(* Logix 5000 project; controller RSL5k_18_Template_noLib Emulate 5570 rev 32.11; software revision 32.02 *)
// Template Application with only task layout pre-installed

TASK _Controller_Status (periodic, rate 250 ms, priority 15, watchdog 2000 ms) : Diagnostics   // L_CPU, etc., and checks for Process Tasks that are Inhibited -- DO NOT INHIBIT THIS TASK
TASK Task_A_50ms (periodic, rate 50 ms, priority 5, watchdog 150 ms) : Task_A_MainProgram   // 50ms period Task
TASK Task_B_100ms (periodic, rate 100 ms, priority 6, watchdog 300 ms) : Task_B_MainProgram   // 100ms period Task
TASK Task_C_250ms (periodic, rate 250 ms, priority 7, watchdog 750 ms) : Task_C_MainProgram   // 250ms period Task
TASK Task_D_500ms (periodic, rate 500 ms, priority 8, watchdog 1500 ms) : Tank1   // 500ms period Task
TASK Task_E_1s (periodic, rate 1000 ms, priority 9, watchdog 3000 ms) : Task_E_MainProgram   // 1000ms (1s) period Task
TASK Task_F_2s (periodic, rate 2000 ms, priority 10, watchdog 6000 ms) : Task_F_MainProgram   // 2000ms (2s) period Task
TASK Task_G_5s (periodic, rate 5000 ms, priority 11, watchdog 15000 ms) : Task_G_MainProgram   // 5000ms (5s) period Task
TASK Task_H_10s (periodic, rate 10000 ms, priority 12, watchdog 30000 ms) : Task_H_MainProgram   // 10000ms (10s) period Task

MODULES
   Local : Emulate 5570 (ICP 2, rev 32.11)
END_MODULES

TYPE P_DescList :   // Code / Description List Entry
STRUCT
   Code : DINT;   // Code for which to look up Description
   Desc : STRING_40;   // Description for given Code
END_STRUCT
END_TYPE

TYPE STRING_12 :
STRUCT
   LEN : DINT;
   DATA : SINT[12];
END_STRUCT
END_TYPE

TYPE STRING_16 :
STRUCT
   LEN : DINT;
   DATA : SINT[16];
END_STRUCT
END_TYPE

TYPE STRING_20 :
STRUCT
   LEN : DINT;
   DATA : SINT[20];
END_STRUCT
END_TYPE

TYPE STRING_40 :
STRUCT
   LEN : DINT;
   DATA : SINT[40];
END_STRUCT
END_TYPE

TYPE STRING_8 :
STRUCT
   LEN : DINT;
   DATA : SINT[8];
END_STRUCT
END_TYPE

TYPE STRING_Area :
STRUCT
   LEN : DINT;
   DATA : SINT[8];
END_STRUCT
END_TYPE

TYPE STRING_Cond :
STRUCT
   LEN : DINT;
   DATA : SINT[20];
END_STRUCT
END_TYPE

TYPE STRING_NavTag :   // Navigation Tag
STRUCT
   LEN : DINT;
   DATA : SINT[20];
END_STRUCT
END_TYPE

ADD_ON_INSTRUCTION JLB_FopdtSim   (* revision 1.0 *)
VAR_INPUT
   cv : REAL; {visible}
   gain : REAL := 1.0; {visible}
   deadTime : REAL := 2.0; {visible}
   timeConst : REAL := 10.0; {visible}
END_VAR
VAR_OUTPUT
   pv : REAL; {access Read Only, visible}
END_VAR
VAR_INPUT
   pvss : REAL; {visible}
   cvss : REAL; {visible}
   pvLimitLow : REAL; {visible}
   pvLimitHigh : REAL := 100.0; {visible}
END_VAR
VAR
   DEDT1 : DEADTIME := (Gain := 1.0, RTSTime := 1);
   LDLG_01 : LEAD_LAG := (Gain := 1.0, RTSTime := 1);
   DEDT1_Array : REAL[500]; {access None}
   SUB_01 : FBD_MATH; {access None}
   HLL_01 : HL_LIMIT; {access None}
   pvUnlimited : REAL; {access None}
   initHigh : REAL; {access None}
   initLow : REAL; {access None}
   LDLG_Limiter_01 : JLB_LdlgLimiter; {access None}
   __l8BF204123A1F2166 : REAL; {access None}
   __l48C57120F21BA85D : REAL; {access None}
   __l0C3A629CB0B0CE2E : REAL; {access None}
   __l3C5358207E677F0D : REAL; {access None}
   __lCAFA7742E4AD4225 : REAL; {access None}
   __lA52B1C482AF3A637 : REAL; {access None}
   __l3430A9F65FF7AABD : REAL; {access None}
   __l4977D2FAECBF782C : REAL; {access None}
   __lBE5B6059D0DA292D : REAL; {access None}
END_VAR

ROUTINE Logic   (* function block diagram *)
   SHEET 1
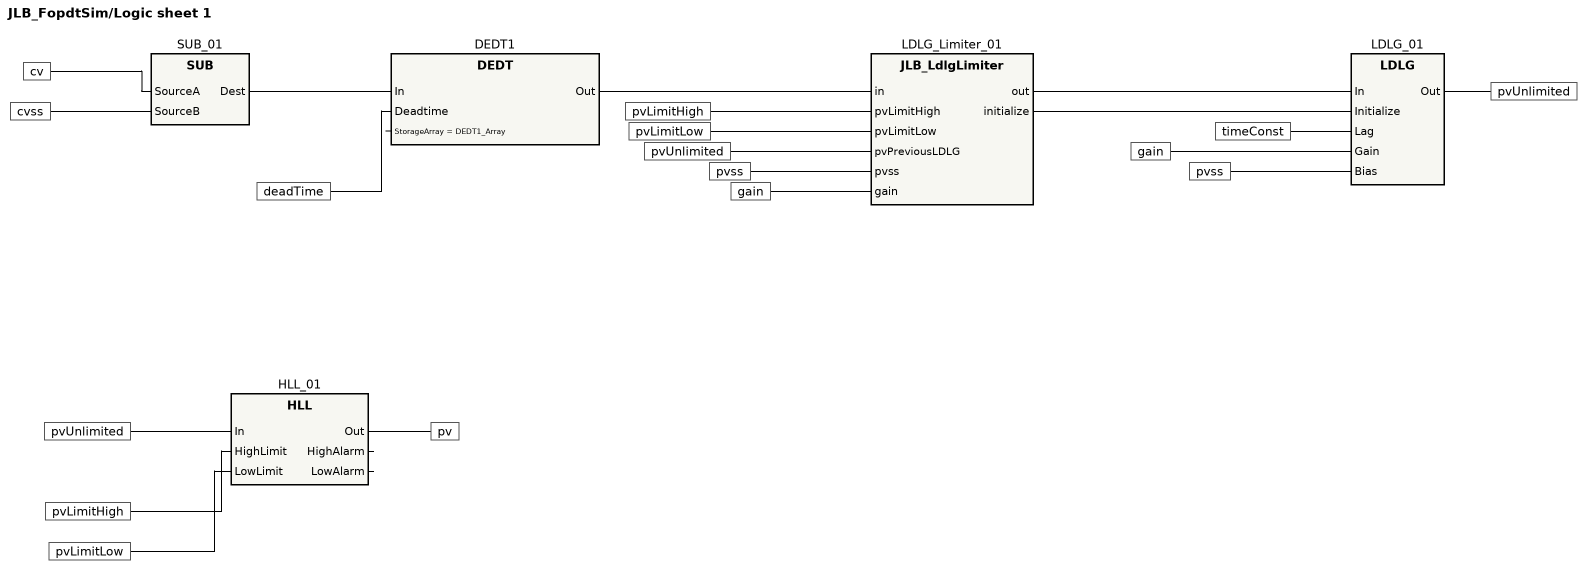
   SUB_01 : SUB(SourceA := cv, SourceB := cvss);
   HLL_01 : HLL(In := pvUnlimited, HighLimit := pvLimitHigh, LowLimit := pvLimitLow);   // unwired pins: HighAlarm LowAlarm
   DEDT1 : DEDT(In := SUB_01.Dest, Deadtime := deadTime, StorageArray := DEDT1_Array);
   pv := HLL_01.Out;
   LDLG_Limiter_01 : JLB_LdlgLimiter(in := DEDT1.Out, pvLimitHigh := pvLimitHigh, pvLimitLow := pvLimitLow, pvPreviousLDLG := pvUnlimited, pvss := pvss, gain := gain);
   LDLG_01 : LDLG(In := LDLG_Limiter_01.out, Initialize := LDLG_Limiter_01.initialize, Lag := timeConst, Gain := gain, Bias := pvss);
   pvUnlimited := LDLG_01.Out;
END_ROUTINE
END_ADD_ON_INSTRUCTION

ADD_ON_INSTRUCTION JLB_IpdtSim   (* revision 1.0 *)
VAR_INPUT
   cv : REAL; {required}
   gain : REAL; {visible}
   deadTime : REAL; {visible}
END_VAR
VAR_OUTPUT
   pv : REAL; {access Read Only, visible}
END_VAR
VAR_INPUT
   cvss : REAL;
   pvLimitHigh : REAL; {visible}
   pvLimitLow : REAL; {visible}
END_VAR
VAR
   DEDT1 : DEADTIME := (Gain := 1.0, RTSTime := 1);
   DEDT1_Array : REAL[500]; {access None}
   SUB_01 : FBD_MATH; {access None}
   INTG_01 : INTEGRATOR := (RTSTime := 1); {access None}
   __lDA04D48D4FBD5F02 : REAL; {access None}
   __lEF2A4DA27C9E24B0 : REAL; {access None}
   __l6744ED6412311BD7 : REAL; {access None}
   __lC3B18D60DF270F58 : REAL; {access None}
   __lFBECCCE1573B33CA : REAL; {access None}
   __lD020E224334B7143 : REAL; {access None}
END_VAR

ROUTINE Logic   (* function block diagram *)
   SHEET 1
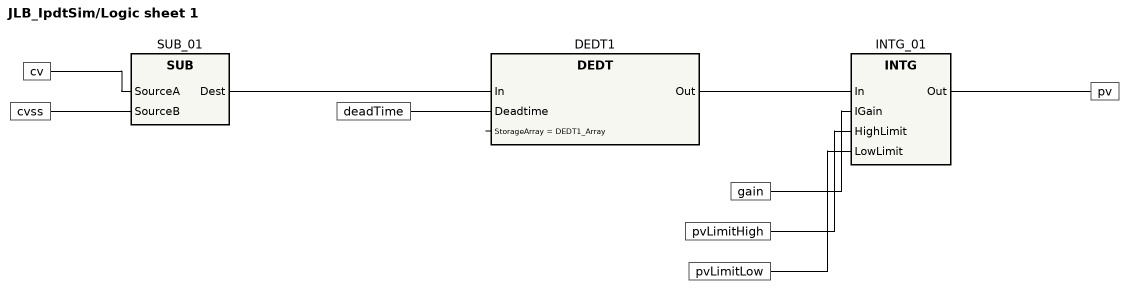
   SUB_01 : SUB(SourceA := cv, SourceB := cvss);
   DEDT1 : DEDT(In := SUB_01.Dest, Deadtime := deadTime, StorageArray := DEDT1_Array);
   INTG_01 : INTG(In := DEDT1.Out, IGain := gain, HighLimit := pvLimitHigh, LowLimit := pvLimitLow);
   pv := INTG_01.Out;
END_ROUTINE
END_ADD_ON_INSTRUCTION

ADD_ON_INSTRUCTION JLB_LdlgLimiter   (* revision 1.0 *)
// Reinitializes a LDLG.Out value to a limit value when limits are exceeded
VAR_INPUT
   in : REAL; {required}   // Normal Process Input
   pvLimitHigh : REAL; {visible}
   pvLimitLow : REAL; {visible}
   pvPreviousLDLG : REAL; {required}   // previous LDLG.Out
   pvss : REAL; {visible}
   gain : REAL; {visible}
END_VAR
VAR_OUTPUT
   out : REAL; {access Read Only, required}   // to LDLG.In
   initialize : BOOL; {access Read Only, visible}   // to LDLG.Initialize
END_VAR
VAR
   initHigh : REAL; {access Read Only}
   initLow : REAL; {access Read Only}
END_VAR

ROUTINE Logic   (* ladder *)
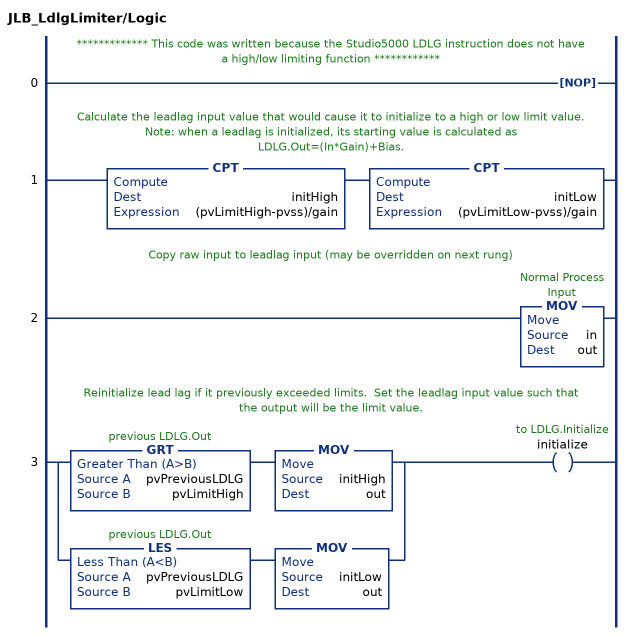
   // ************* This code was written because the Studio5000 LDLG instruction does not have a high/low limiting function ************
   0: NOP();
   // Calculate the leadlag input value that would cause it to initialize to a high or low limit value.
   // Note: when a leadlag is initialized, its starting value is calculated as LDLG.Out=(In*Gain)+Bias.
   1: CPT(initHigh,(pvLimitHigh-pvss)/gain)CPT(initLow,(pvLimitLow-pvss)/gain);
   // Copy raw input to leadlag input (may be overridden on next rung)
   2: MOV(in,out);
   // Reinitialize lead lag if it previously exceeded limits.  Set the leadlag input value such that the output will be the limit value.
   3: [GRT(pvPreviousLDLG,pvLimitHigh) MOV(initHigh,out) ,LES(pvPreviousLDLG,pvLimitLow) MOV(initLow,out) ]OTE(initialize);
END_ROUTINE
END_ADD_ON_INSTRUCTION

ADD_ON_INSTRUCTION L_TaskMon   (* revision 4.10 .00 Release, vendor Rockwell Automation *)
// Logix Task Monitor
// Revision note:
// See Instruction Help for a summary of changes, and see 4.10 Release Notes for details.
// Help:
// Copyright © Rockwell Automation, Inc.  All Rights Reserved.
// This Instruction monitors the controller Task in which it is contained and provides:
// *  Display Values for Task configuration: Task Name, Priority, Rate, Watchdog settings
// *  Display Values for Task statistics: Last and Max Execution time, Overlap Count
// *  Display of the Task Inhibit / Active Status
// *  Configuration of a "Plan" Execution Time, the time in which the Task is expected
//      to always complete (including interrupts by higher priority Tasks)
// *  An optional Alarm when Last (actual) Execution Time exceeds Plan
// *  A Reset command, which clears and acknowledges the Over Plan Alarm.
// *  Maintenance Commands to clear the Max Execution Time and Overlap Count.
// *  A configurable single-letter Task Identifier (for HMI)
// SUMMARY OF CHANGES FROM PREVIOUS VERSION (4.00.00)
// See 4.10 Release Notes for details.
// * Unmodified, up-rev only for Library 4.10.00
// SUMMARY OF CHANGES FROM PREVIOUS VERSION (3.5-01)
// See 4.00 Release Notes for details.
// * Changed Inf_ items to HMI_, and added Cfg_Area for security.
// * Deleted Cfg_PCmdClear; all Program Commands are now self-clearing.
// * Aligned ready bit naming with command bit names.
// * Removed unused STRING Local Tags.
// * All OCmds/MCmds and ORdys/MRdys are now Local Tags.
// * Added Sts_RdyAck and Sts_RdyReset for use by external objects.
VAR_INPUT
   Inp_Reset : BOOL; {visible}   // 1=Reset Max Task Time and any Alarm requiring reset
   Cfg_HasOverPlanAlm : ALIAS FOR OverPlan.Cfg_Exists;   // 1=Task Plan Exceeded Alarm exists and will be checked
   Cfg_OverPlanResetReqd : ALIAS FOR OverPlan.Cfg_ResetReqd;   // 1=Task Plan Exceeded Alarm is latched in, requires Reset Command to clear
   Cfg_OverPlanAckReqd : ALIAS FOR OverPlan.Cfg_AckReqd;   // 1=Task Plan Exceeded Alarm must be acknowledged
   Cfg_OverPlanSeverity : ALIAS FOR OverPlan.Cfg_Severity;   // Task Plan Exceeded Alarm Severity: 1=low, 2=medium, 3=high, 4=highest
   Cfg_PlanExecT : REAL := 3000.0;   // Expected Execution Time of Task (including interrupts) (ms)
   PCmd_Reset : BOOL;   // Program Command to Reset latched Alarm and Max Task Time
   PCmd_OverPlanAck : ALIAS FOR OverPlan.PCmd_Reset;   // Program Command to Acknowledge the Task Plan Exceeded Alarm
   PCmd_OverPlanSuppress : ALIAS FOR OverPlan.PCmd_Suppress;   // Program Command to Inhibit the Task Plan Exceeded Alarm
   PCmd_OverPlanUnsuppress : ALIAS FOR OverPlan.PCmd_Unsuppress;   // Program Command to Uninhibit the Task Plan Exceeded Alarm
   PCmd_OverPlanUnshelve : ALIAS FOR OverPlan.PCmd_Unshelve;   // Program Command to Unshelve the Task Plan Exceeded Alarm
END_VAR
VAR_OUTPUT
   Val_Rate : REAL; {access Read Only, visible}   // Configured Task Period (ms)
   Val_Priority : DINT; {access Read Only, visible}   // Configured Task Priority (1..15, lower number is higher priority)
   Val_LastExecT : REAL; {access Read Only, visible}   // Actual Last Execution Time of Task (ms)
   Val_MaxExecT : REAL; {access Read Only, visible}   // Highest Execution Time of Task (ms)
   Val_OverlapC : DINT; {access Read Only, visible}   // Task Overlap Count
   Val_WatchdogT : REAL; {access Read Only, visible}   // Configured Task Watchdog Timer Value (ms)
   Val_NotifyAll : DINT; {access Read Only}   // Highest Alarm prio and ack status this object + channel (enum)
   Val_UnackAlmC : DINT; {access Read Only}   // Count of Unacknowledged Alarms
   Sts_TaskInhibited : BOOL; {access Read Only, visible}   // 1=Task is Inhibited, 0 = Task is Active
   Sts_AlmInh : BOOL; {access Read Only}   // 1=An Alarm is Shelved, Disabled or Suppressed: display icon
   Sts_Err : BOOL; {access Read Only, visible}   // 1=Error in Config: see detail bits for reason
   Err_Plan : BOOL; {access Read Only}   // 1=Error in Config: Task Planned Exec Time (use 0.1 to 20,000.0 ms)
   Err_Alarm : BOOL; {access Read Only}   // 1=Error in Config: Alarm Min On Time or Severity
   Sts_RdyReset : ALIAS FOR ORdy_Reset; {access Read Only}   // 1=A latched alarm or shed condition is ready to be reset
   Sts_RdyAck : BOOL; {access Read Only}   // 1=An alarm is ready to be acknowledged
   Sts_OverPlan : ALIAS FOR OverPlan.Inp; {visible}   // 1=Task Actual Time exceeds Plan Time
   Alm_OverPlan : ALIAS FOR OverPlan.Alm;   // 1=Alarm: Planned Task Time Exceeded
   Ack_OverPlan : ALIAS FOR OverPlan.Ack;   // 1=Task Plan Exceeded Alarm has been acknowledged
   Sts_OverPlanDisabled : ALIAS FOR OverPlan.Disabled;   // 1=Task Plan Exceeded Alarm has been Disabled by Maintenance
   Sts_OverPlanSuppressed : ALIAS FOR OverPlan.Suppressed;   // 1=Task Plan Exceeded Alarm has been Suppressed by Program
   Sts_OverPlanShelved : ALIAS FOR OverPlan.Shelved;   // 1=Task Plan Exceeded Alarm has been Shelved by Operator
   L_TaskMon : BOOL;   // Unique Parameter Name for auto - discovery
END_VAR
VAR
   OverPlan : P_Alarm := (Inp := 1, Cfg_Exists := 1, Cfg_AckReqd := 1, Cfg_AllowShelve := 1, Cfg_AllowDisable := 1, Cfg_Severity := 750, Cfg_AlmMinOnT := 5, PCfg_AllowExist := 1, Ack := 1);   // Alarm if Actual Task Execution Time exceeds Planned
   Wrk_Inhibited : DINT; {access None}   // Task Inhibited if nonzero, Active if zero
   Val_Name : STRING_40; {access Read Only}   // Task Name as configured in Controller
   Wrk_Rate : DINT; {access None}   // Task Configured Rate (Period) from GSV (us)
   Wrk_LastExecT : DINT; {access None}   // Task Last Execution Time from GSV (us)
   Wrk_MaxExecT : DINT; {access None}   // Task Maximum Execution Time from GSV (us)
   Wrk_WatchdogT : DINT; {access None}   // Task Configured Watchdog Time from GSV (us)
   HMI_Tab : SINT;   // Tab to display (FTView ME)
   Wrk_Notify : DINT; {access None}   // Buffer for building Val_Notify
   Val_Notify : DINT; {access Read Only}   // Current Alarm Level and Acknowledgement (enumeration)
   HMI_Type : STRING_16 := 'L_TaskMon'; {access Read Only}   // Must contain AOI name, used for HMI and Information S/W
   Cfg_Area : STRING_Area := 'area01';   // Process Area for security
   HMI_Lib : STRING_12 := 'RA-BAS'; {access Read Only}   // Display Library for Faceplate call-up
   Wrk_UnackAlmC : DINT; {access None}   // Buffer for building Val_UnackAlmC
   ORdy_ResetAckAll : BOOL; {access Read Only}   // 1=At least one Alarm requires Reset or Acknowledgement
   ORdy_Reset : BOOL; {access Read Only}   // 1=Ready for OCmd_Reset (enables button)
   OCmd_ResetAckAll : BOOL;   // Operator Command to Reset and Acknowledge all Alarms
   OCmd_Reset : BOOL;   // Operator Command to Reset latched Alarm and Max Task Time
   MCmd_ClearOverlapC : BOOL;   // Maintenance Command to Clear Task Overlap Count
   MCmd_ClearMaxExecT : BOOL;   // Maintenance Command to Clear Maximum Execution Time
END_VAR

ROUTINE Logic   (* ladder *)
// Monitor the Task containing this AOI and alarm if over planned scan time.
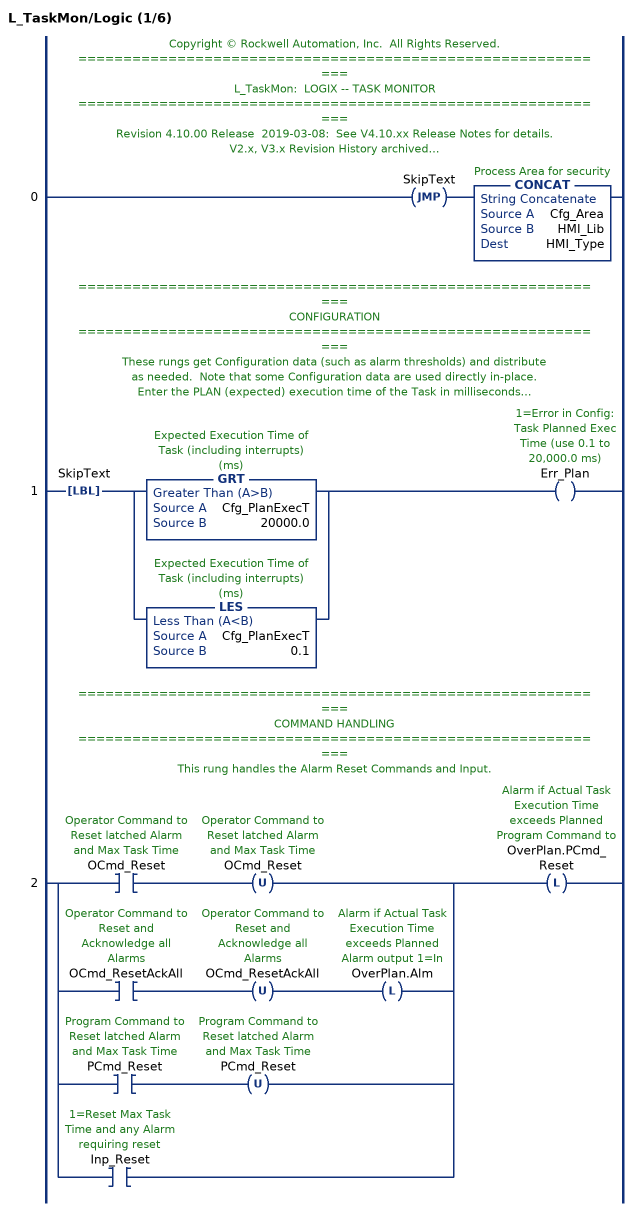
   // Copyright © Rockwell Automation, Inc.  All Rights Reserved.
   // ============================================================
   // L_TaskMon:  LOGIX -- TASK MONITOR
   // ============================================================
   // Revision 4.10.00 Release  2019-03-08:  See V4.10.xx Release Notes for details.
   // V2.x, V3.x Revision History archived.
   // V4.00.00  2018-06-19:  Changed Inf_ items to HMI_ and added Cfg_Area for security.
   // Added unacked alarm count. Deleted Cfg_PCmdClear; all Program
   // Commands are now self-clearing. Aligned ready bit naming with
   // command bit names. Removed unused STRING Local Tags.
   // All OCmds/MCmds and ORdys/MRdys are now Local Tags.
   // Added Sts_RdyAck and Sts_ResetReqd for use by external objects.
   // V4.10.00  2019-03-08:  Unmodified, up-rev only for Library 4.10.00
   // ============================================================
   // This Instruction monitors the controller Task in which it is contained
   // and provides:
   // *  Display Values for Task configuration: Task Name, Priority, Rate, Watchdog settings
   // *  Display Values for Task statistics: Last and Max Execution time, Overlap Count
   // *  Display of the Task Inhibit / Active Status
   // *  Configuration of a "Plan" Execution Time, the time in which the Task is expected
   //  to always complete (including interrupts by higher priority Tasks)
   // *  An optional Alarm when Last (actual) Execution Time exceeds Plan
   // *  A Reset command, which clears and acknowledges the Over Plan Alarm.
   // *  Maintenance Commands to clear the Max Execution Time and Overlap Count.
   // *  A configurable single-letter Task Identifier (for HMI)
   // ============================================================
   // SHOW LOCAL STRINGS
   // ============================================================
   // The STRINGs containing the text associated with each instance of this
   // instruction cannot be Input or Output Parameters, because STRINGs are not
   //  'atomic' types. (Inputs and Outputs must be SINT, INT, DINT, REAL, or BOOL.)
   // In order to make it easier to find and configure these STRINGs, this rung
   // was added.  THE JMP (and the LBL on the following rung)
   // MUST NOT BE REMOVED!!!
   // To view the STRINGs, go to the instruction instance (in LD or FBD), RIGHT-click
   // to bring up the context menu and select "Open Instruction Logic".
   // This rung will appear with the STRING values for the selected instance.
   // You may double-click the STRING values here to modify them as well.
   // #####  V4.00.00  2018-06-19:  Added string for Cfg_Area, renamed Inf_* to HMI_*,  #####
   // #####  removed unused STRING Local Tags.  #####
   0: JMP(SkipText)CONCAT(Cfg_Area,HMI_Lib,HMI_Type);
   // ============================================================
   // CONFIGURATION
   // ============================================================
   // These rungs get Configuration data (such as alarm thresholds) and distribute
   // as needed.  Note that some Configuration data are used directly in-place.
   // Enter the PLAN (expected) execution time of the Task in milliseconds.
   // If the actual execution time of the Task (which includes interrupts by higher priority
   // Tasks) exceeds this threshold, the OverPlan Status is raised
   // (and the OverPlan Alarm is raised if so configured).
   1: LBL(SkipText)[GRT(Cfg_PlanExecT,20000.0) ,LES(Cfg_PlanExecT,0.1) ]OTE(Err_Plan);
   // ============================================================
   // COMMAND HANDLING
   // ============================================================
   // This rung handles the Alarm Reset Commands and Input.
   2: [XIC(OCmd_Reset) OTU(OCmd_Reset) ,XIC(OCmd_ResetAckAll) OTU(OCmd_ResetAckAll) OTL(OverPlan.Alm) ,XIC(PCmd_Reset) OTU(PCmd_Reset) ,XIC(Inp_Reset) ]OTL(OverPlan.PCmd_Reset);
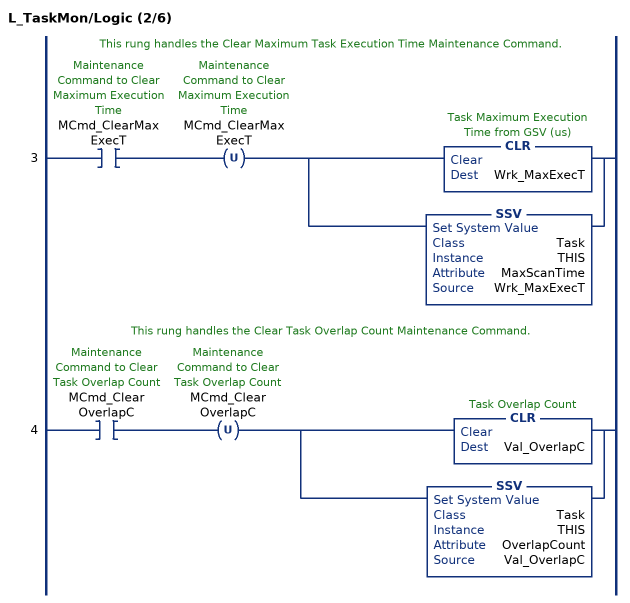
   // This rung handles the Clear Maximum Task Execution Time Maintenance Command.
   3: XIC(MCmd_ClearMaxExecT)OTU(MCmd_ClearMaxExecT)[CLR(Wrk_MaxExecT) ,SSV(Task,THIS,MaxScanTime,Wrk_MaxExecT) ];
   // This rung handles the Clear Task Overlap Count Maintenance Command.
   4: XIC(MCmd_ClearOverlapC)OTU(MCmd_ClearOverlapC)[CLR(Val_OverlapC) ,SSV(Task,THIS,OverlapCount,Val_OverlapC) ];
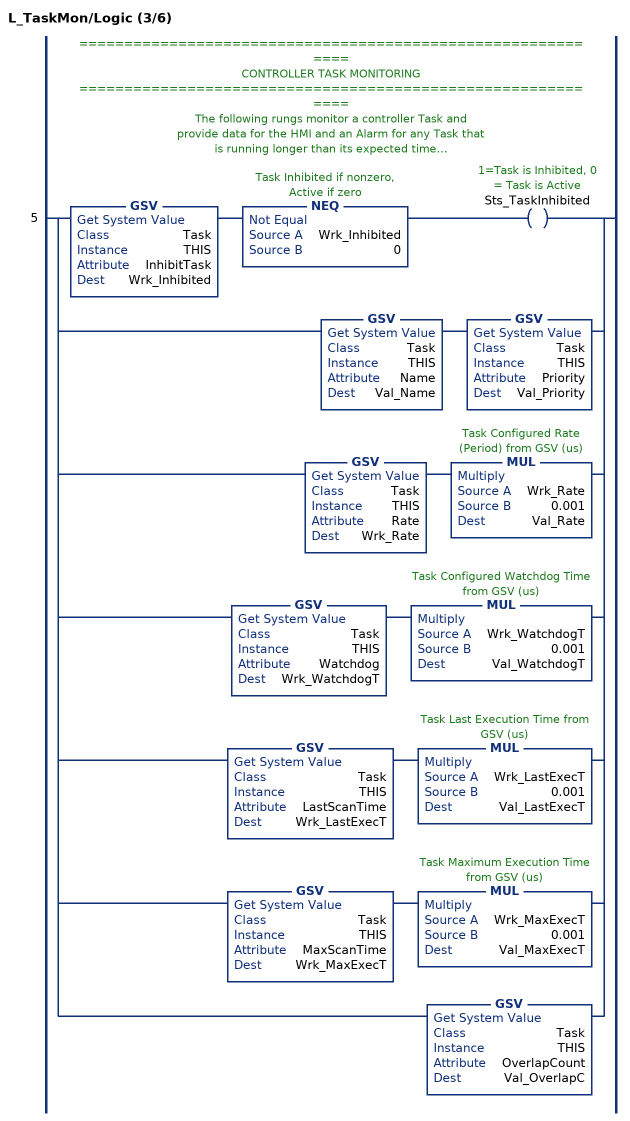
   // ============================================================
   // CONTROLLER TASK MONITORING
   // ============================================================
   // The following rungs monitor a controller Task and
   // provide data for the HMI and an Alarm for any Task that
   // is running longer than its expected time.
   // This rung provides the following Task configuration data:
   // * Task Inhibited status
   // * Task Name
   // * Task Priority
   // * Task Period (Rate) (ms)
   // * Task Watchdog Timeout setting (ms)
   // ... and provides the following Task statistics:
   // * Task Last Execution Time (ms)
   // * Task Maximum Execution Time (ms)
   // * Task Overlap Count
   5: [GSV(Task,THIS,InhibitTask,Wrk_Inhibited) NEQ(Wrk_Inhibited,0) OTE(Sts_TaskInhibited) ,GSV(Task,THIS,Name,Val_Name) GSV(Task,THIS,Priority,Val_Priority) ,GSV(Task,THIS,Rate,Wrk_Rate) MUL(Wrk_Rate,0.001,Val_Rate) ,GSV(Task,THIS,Watchdog,Wrk_WatchdogT) MUL(Wrk_WatchdogT,0.001,Val_WatchdogT) ,GSV(Task,THIS,LastScanTime,Wrk_LastExecT) MUL(Wrk_LastExecT,0.001,Val_LastExecT) ,GSV(Task,THIS,MaxScanTime,Wrk_MaxExecT) MUL(Wrk_MaxExecT,0.001,Val_MaxExecT) ,GSV(Task,THIS,OverlapCount,Val_OverlapC) ];
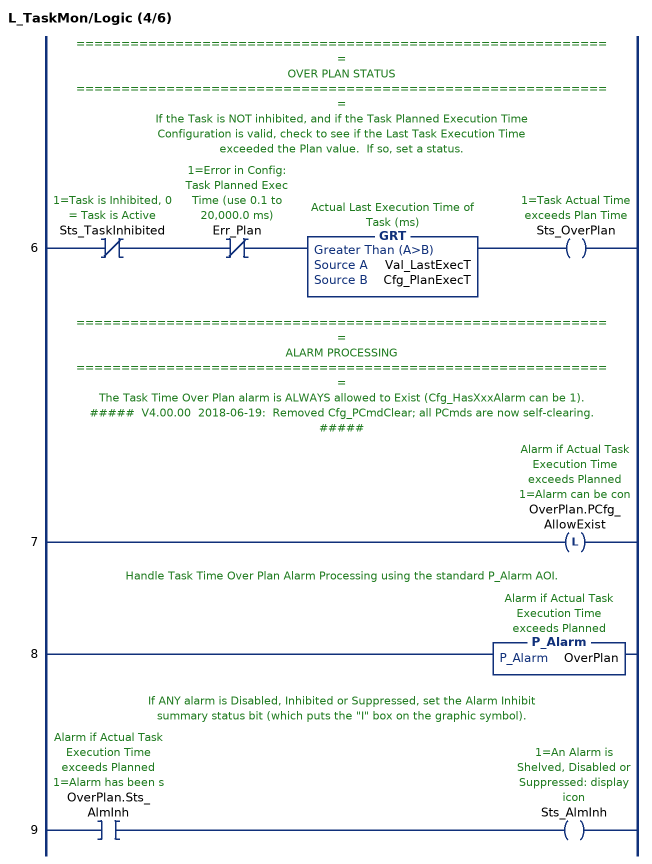
   // ============================================================
   // OVER PLAN STATUS
   // ============================================================
   // If the Task is NOT inhibited, and if the Task Planned Execution Time
   // Configuration is valid, check to see if the Last Task Execution Time
   // exceeded the Plan value.  If so, set a status.
   6: XIO(Sts_TaskInhibited)XIO(Err_Plan)GRT(Val_LastExecT,Cfg_PlanExecT)OTE(Sts_OverPlan);
   // ============================================================
   // ALARM PROCESSING
   // ============================================================
   // The Task Time Over Plan alarm is ALWAYS allowed to Exist (Cfg_HasXxxAlarm can be 1).
   // #####  V4.00.00  2018-06-19:  Removed Cfg_PCmdClear; all PCmds are now self-clearing.  #####
   7: OTL(OverPlan.PCfg_AllowExist);
   // Handle Task Time Over Plan Alarm Processing using the standard P_Alarm AOI.
   8: P_Alarm(OverPlan);
   // If ANY alarm is Disabled, Inhibited or Suppressed, set the Alarm Inhibit
   // summary status bit (which puts the "I" box on the graphic symbol).
   9: XIC(OverPlan.Sts_AlmInh)OTE(Sts_AlmInh);
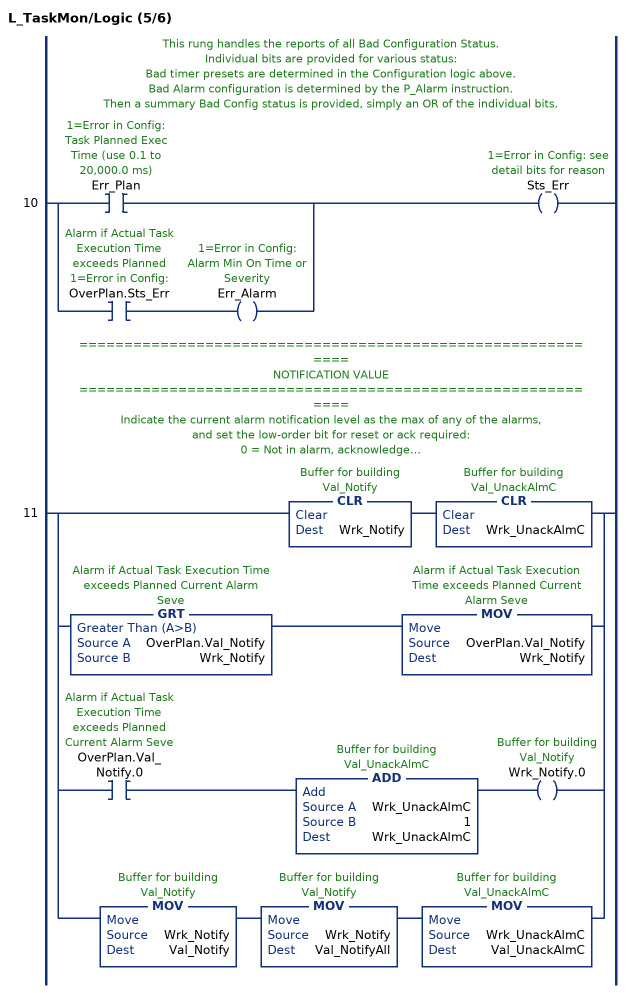
   // This rung handles the reports of all Bad Configuration Status.
   // Individual bits are provided for various status:
   // Bad timer presets are determined in the Configuration logic above.
   // Bad Alarm configuration is determined by the P_Alarm instruction.
   // Then a summary Bad Config status is provided, simply an OR of the individual bits.
   10: [XIC(Err_Plan) ,XIC(OverPlan.Sts_Err) OTE(Err_Alarm) ]OTE(Sts_Err);
   // ============================================================
   // NOTIFICATION VALUE
   // ============================================================
   // Indicate the current alarm notification level as the max of any of the alarms,
   // and set the low-order bit for reset or ack required:
   // 0 = Not in alarm, acknowledged
   // 1 = Not in alarm, unacknowledged or reset required
   // 2 = Low severity alarm, acknowledged
   // 3 = Low severity alarm, unacknowledged
   // 4 = Medium severity alarm, acknowledged
   // 5 = Medium severity alarm, unacknowledged
   // 6 = High severity alarm, acknowledged
   // 7 = High severity alarm, unacknowledged
   // 8 = Urgent severity alarm, acknowledged
   // 9 = Urgent severity alarm, unacknowledged
   // #####  V4.00.00  2018-06-19:  Added Val_NotifyAll and unacked alarm count.  #####
   11: [CLR(Wrk_Notify) CLR(Wrk_UnackAlmC) ,GRT(OverPlan.Val_Notify,Wrk_Notify) MOV(OverPlan.Val_Notify,Wrk_Notify) ,XIC(OverPlan.Val_Notify.0) ADD(Wrk_UnackAlmC,1,Wrk_UnackAlmC) OTE(Wrk_Notify.0) ,MOV(Wrk_Notify,Val_Notify) MOV(Wrk_Notify,Val_NotifyAll) MOV(Wrk_UnackAlmC,Val_UnackAlmC) ];
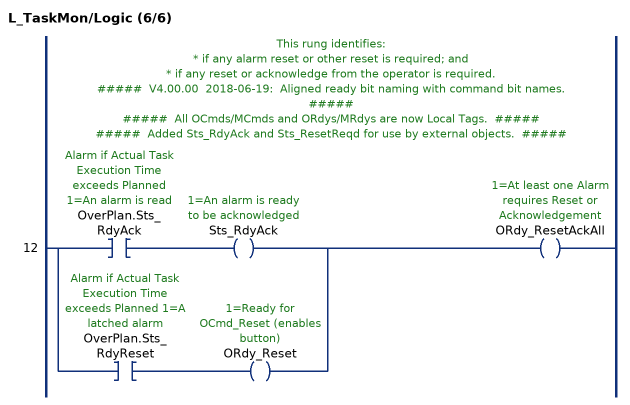
   // This rung identifies:
   // * if any alarm reset or other reset is required; and
   // * if any reset or acknowledge from the operator is required.
   // #####  V4.00.00  2018-06-19:  Aligned ready bit naming with command bit names.  #####
   // #####  All OCmds/MCmds and ORdys/MRdys are now Local Tags.  #####
   // #####  Added Sts_RdyAck and Sts_ResetReqd for use by external objects.  #####
   12: [XIC(OverPlan.Sts_RdyAck) OTE(Sts_RdyAck) ,XIC(OverPlan.Sts_RdyReset) OTE(ORdy_Reset) ]OTE(ORdy_ResetAckAll);
END_ROUTINE
END_ADD_ON_INSTRUCTION

ADD_ON_INSTRUCTION P_AIn   (* revision 4.10 .00 Release, vendor Rockwell Automation, ExecutePrescan, ExecuteEnableInFalse *)
// Analog Input
// Revision note:
// See Instruction Help for a summary of changes, and see 4.10 Release Notes for details.
// Help:
// Copyright © Rockwell Automation, Inc.  All Rights Reserved.
// This Instruction monitors an Analog Input from a flow, level, pressure,
// temperature, or any other analog sensor, and provides:
// *  Scaling, from Input (Raw) to PV (Engineering) Units
// *  High-High, High, Low and Low-Low Status and Alarms, with Gate
// inputs and configurable on-delay, off-delay and gate delay times
// *  Monitoring of bad/uncertain PV status, floating point exceptions
// and out-of-range conditions, with PV Fail alarm
// *  Setting of a simulated input signal for process simulation
// *  Capturing of the lowest and highest PV excursion values
// *  Configuration for status thresholds, deadbands and range limits
// *  Maintenance Commands to allow manual override of the input signal (Substitute PV)
// Alarms are provided by P_Alarm AOI instances.
// Status gating provided by P_Gate AOI instances.
// SUMMARY OF CHANGES FROM PREVIOUS VERSION (4.00.01)
// See 4.10 Release Notes for details.
// * Added Cfg_HasMoreObj.
// SUMMARY OF CHANGES FROM PREVIOUS VERSION (4.00.00)
// See 4.00 Release Notes for details.
// * Modified handling of SrcQ_IO and SrcQ.
// SUMMARY OF CHANGES FROM PREVIOUS VERSION (3.5-03)
// See 4.00 Release Notes for details.
// * Removed P_Mode, PSet/Val_Owner and related OSets,
//    PSets and Vals.  Thresholds are now Cfgs.
// * Changed Inf_ items to HMI_, and added Cfg_Area for security.
// * Added notify and unack count rollup for Channel object.
// * Changed Out-of-Range limit checks to use raw Input (Inp_PV)
//    instead of scaled PV (Val).  Changing EU scaling will not
//    necessitate changing fail thresholds and deadband.
// * Deleted Cfg_PCmdClear.  All Program Commands are now self-clearing.
// * Aligned ready bit naming with command bit names.
// * All OCmds/MCmds and ORdys/MRdys are now Local Tags.
// * Added Sts_RdyAck and Sts_RdyReset for use by external objects.
// * Removed Err_DB, code ensures Status Deadband configs are always valid.
// * Added configurable decimal places for display on HMI.
VAR_INPUT
   Inp_PV : REAL; {visible}   // Input Signal (process variable) from Sensor
   Inp_PVSrcQ : DINT;   // Input Source and Quality (from Channel object, if available) (enum)
   Inp_PVNotify : DINT;   // Related PV object alarm prio and ack status (enum)
   Inp_PVBad : BOOL;   // 1=PV or I/O Comms Status Bad, 0=OK
   Inp_PVUncertain : BOOL;   // 1=PV Value Not Reliable, 0=OK
   Inp_Sim : BOOL;   // 1=Use simulated PV (Set_SimPV); 0=Use Input (Inp_PV)
   Inp_HiHiGate : ALIAS FOR HiHiGate.Inp_Gate;   // High-High Status Gate, 1=enabled
   Inp_HiGate : ALIAS FOR HiGate.Inp_Gate;   // High Status Gate, 1=enabled
   Inp_LoGate : ALIAS FOR LoGate.Inp_Gate;   // Low Status Gate, 1=enabled
   Inp_LoLoGate : ALIAS FOR LoLoGate.Inp_Gate;   // Low-Low Status Gate, 1=enabled
   Inp_FailGate : ALIAS FOR FailGate.Inp_Gate;   // Fail Status Gate, 1=enabled
   Inp_Reset : BOOL;   // 1=Reset all Alarms requiring reset
   Cfg_NoSubstPV : BOOL;   // 1=Disallow selection of Substitute PV
   Cfg_HasChanObj : BOOL;   // 1=Tells HMI a Channel object (AIChan, etc.) is used for Inp_PV
   Cfg_HasMoreObj : BOOL;   // 1=Tells HMI an object with more info is available
   Cfg_UseChanSrcQ : BOOL;   // 1=Pass thru connected Channel's SrcQ value, 0=generate SrcQ
   Cfg_PVDecPlcs : DINT := 2;   // Number of decimal places for PV display (0..6)
   Cfg_HasHiHiAlm : ALIAS FOR HiHi.Cfg_Exists;   // 1=High-High Alarm exists and will be checked
   Cfg_HasHiAlm : ALIAS FOR Hi.Cfg_Exists;   // 1=High Alarm exists and will be checked
   Cfg_HasLoAlm : ALIAS FOR Lo.Cfg_Exists;   // 1=Low Alarm exists and will be checked
   Cfg_HasLoLoAlm : ALIAS FOR LoLo.Cfg_Exists;   // 1=Low-Low Alarm exists and will be checked
   Cfg_HasFailAlm : ALIAS FOR Fail.Cfg_Exists;   // 1=Analog Input Failure Alarm exists and will be checked
   Cfg_HiHiResetReqd : ALIAS FOR HiHi.Cfg_ResetReqd;   // 1=Reset required to clear High-High Alarm
   Cfg_HiResetReqd : ALIAS FOR Hi.Cfg_ResetReqd;   // 1=Reset required to clear High Alarm
   Cfg_LoResetReqd : ALIAS FOR Lo.Cfg_ResetReqd;   // 1=Reset required to clear Low Alarm
   Cfg_LoLoResetReqd : ALIAS FOR LoLo.Cfg_ResetReqd;   // 1=Reset required to clear Low-Low Alarm
   Cfg_FailResetReqd : ALIAS FOR Fail.Cfg_ResetReqd;   // 1=Reset required to clear Analog InputFailure Alarm
   Cfg_HiHiAckReqd : ALIAS FOR HiHi.Cfg_AckReqd;   // 1=Acknowledge required for High-High Alarm
   Cfg_HiAckReqd : ALIAS FOR Hi.Cfg_AckReqd;   // 1=Acknowledge required for High Alarm
   Cfg_LoAckReqd : ALIAS FOR Lo.Cfg_AckReqd;   // 1=Acknlowledge required for Low Alarm
   Cfg_LoLoAckReqd : ALIAS FOR LoLo.Cfg_AckReqd;   // 1=Acknowledge required for Low-Low Alarm
   Cfg_FailAckReqd : ALIAS FOR Fail.Cfg_AckReqd;   // 1=Acknowledge required for Analog Input Failure Alarm
   Cfg_HiHiSeverity : ALIAS FOR HiHi.Cfg_Severity;   // High-High Alarm Severity: 1..250=Low, 251..500=Medium, 501..750=High, 751..1000=Urgent
   Cfg_HiSeverity : ALIAS FOR Hi.Cfg_Severity;   // High Alarm Severity: 1..250=Low, 251..500=Medium, 501..750=High, 751..1000=Urgent
   Cfg_LoSeverity : ALIAS FOR Lo.Cfg_Severity;   // Low Alarm Severity: 1..250=Low, 251..500=Medium, 501..750=High, 751..1000=Urgent
   Cfg_LoLoSeverity : ALIAS FOR LoLo.Cfg_Severity;   // Low-Low Alarm Severity: 1..250=Low, 251..500=Medium, 501..750=High, 751..1000=Urgent
   Cfg_FailSeverity : ALIAS FOR Fail.Cfg_Severity;   // Failure Alarm Severity: 1..250=Low, 251..500=Medium, 501..750=High, 751..1000=Urgent
   Cfg_InpRawMin : REAL;   // Input (unscaled) Minimum for Scaling
   Cfg_InpRawMax : REAL := 100.0;   // Input (unscaled) Maximum for Scaling
   Cfg_PVEUMin : REAL;   // PV (Output) Minimum for Scaling to EU
   Cfg_PVEUMax : REAL := 100.0;   // PV (Output) Maximum for Scaling to EU
   Cfg_FiltTC : REAL;   // PV Filter Time Constant (s), 0.0 = unfiltered
   Cfg_HiHiLim : REAL := 1.5e+38; {visible}   // High-High Status Threshold (EU)
   Cfg_HiHiDB : REAL := 1.0;   // High-High Status Deadband (EU)
   Cfg_HiHiOnDly : ALIAS FOR HiHiGate.Cfg_OnDly;   // Minimum time above High-High Limit to raise Status (s)
   Cfg_HiHiOffDly : ALIAS FOR HiHiGate.Cfg_OffDly;   // Minimum time below High-High Limit (minus deadband) to clear Status (s)
   Cfg_HiHiGateDly : ALIAS FOR HiHiGate.Cfg_GateDly;   // High-High Status Gate Delay (s)
   Cfg_HiLim : REAL := 1.5e+38; {visible}   // High Status Threshold (EU)
   Cfg_HiDB : REAL := 1.0;   // High Status Deadband (EU)
   Cfg_HiOnDly : ALIAS FOR HiGate.Cfg_OnDly;   // Minimum time above High Limit to raise Status (s)
   Cfg_HiOffDly : ALIAS FOR HiGate.Cfg_OffDly;   // Minimum time below High Limit (minus deadband) to clear Status (s)
   Cfg_HiGateDly : ALIAS FOR HiGate.Cfg_GateDly;   // High Status Gate Delay (s)
   Cfg_LoLim : REAL := -1.5e+38; {visible}   // Low Status Threshold (EU)
   Cfg_LoDB : REAL := 1.0;   // Low Status Deadband (EU)
   Cfg_LoOnDly : ALIAS FOR LoGate.Cfg_OnDly;   // Minimum time below Low Limit to raise Status (s)
   Cfg_LoOffDly : ALIAS FOR LoGate.Cfg_OffDly;   // Minimum time above Low Limit (plus deadband) to clear Status (s)
   Cfg_LoGateDly : ALIAS FOR LoGate.Cfg_GateDly;   // Low Status Gate Delay (s)
   Cfg_LoLoLim : REAL := -1.5e+38; {visible}   // Low-Low Status Threshold (EU)
   Cfg_LoLoDB : REAL := 1.0;   // Low-Low Status Deadband (EU)
   Cfg_LoLoOnDly : ALIAS FOR LoLoGate.Cfg_OnDly;   // Minimum time below Low-Low Limit to raise Status (s)
   Cfg_LoLoOffDly : ALIAS FOR LoLoGate.Cfg_OffDly;   // Minimum time above Low-Low Limit (plus deadband) to clear Status (s)
   Cfg_LoLoGateDly : ALIAS FOR LoLoGate.Cfg_GateDly;   // Low-Low Status Gate Delay (s)
   Cfg_FailHiLim : REAL := 103.958336;   // Out-of-Range (fail) High Limit (raw units)
   Cfg_FailLoLim : REAL := -2.0833333;   // Out-of-Range (fail) Low Limit (raw units)
   Cfg_FailDB : REAL := 0.41666666;   // Out-of-Range (fail) High/Low Deadband (raw units)
   Cfg_FailOnDly : ALIAS FOR FailGate.Cfg_OnDly;   // Minimum time Bad or Out of Range to raise Fail Status (s)
   Cfg_FailOffDly : ALIAS FOR FailGate.Cfg_OffDly;   // Minimum time OK or In Range to clear Fail Status (s)
   Cfg_FailGateDly : ALIAS FOR FailGate.Cfg_GateDly;   // Fail Status Gate Delay (s)
   Set_SimPV : REAL;   // PV used in Simulation (Inp_Sim=1) (EU)
   PCmd_ClearCapt : BOOL;   // Program Command to Clear the captured min / max PV excursion values
   PCmd_Reset : BOOL;   // Program Command to Reset all Alarms requiring Reset
   PCmd_HiHiAck : ALIAS FOR HiHi.PCmd_Ack;   // Program Command to Acknowledge High-High Alarm
   PCmd_HiHiSuppress : ALIAS FOR HiHi.PCmd_Suppress;   // Program Command to Suppress High-High Alarm
   PCmd_HiHiUnsuppress : ALIAS FOR HiHi.PCmd_Unsuppress;   // Program Command to Unsuppress High-High Alarm
   PCmd_HiHiUnshelve : ALIAS FOR HiHi.PCmd_Unshelve;   // Program Command to Unshelve High-High Alarm
   PCmd_HiAck : ALIAS FOR Hi.PCmd_Ack;   // Program Command to Acknowledge High Alarm
   PCmd_HiSuppress : ALIAS FOR Hi.PCmd_Suppress;   // Program Command to Suppress High Alarm
   PCmd_HiUnsuppress : ALIAS FOR Hi.PCmd_Unsuppress;   // Program Command to Unsuppress High Alarm
   PCmd_HiUnshelve : ALIAS FOR Hi.PCmd_Unshelve;   // Program Command to Unshelve High Alarm
   PCmd_LoAck : ALIAS FOR Lo.PCmd_Ack;   // Program Command to Acknowledge Low Alarm
   PCmd_LoSuppress : ALIAS FOR Lo.PCmd_Suppress;   // Program Command to Suppress Low Alarm
   PCmd_LoUnsuppress : ALIAS FOR Lo.PCmd_Unsuppress;   // Program Command to Unsuppress Low Alarm
   PCmd_LoUnshelve : ALIAS FOR Lo.PCmd_Unshelve;   // Program Command to Unshelve Low Alarm
   PCmd_LoLoAck : ALIAS FOR LoLo.PCmd_Ack;   // Program Command to Acknowledge Low-Low Alarm
   PCmd_LoLoSuppress : ALIAS FOR LoLo.PCmd_Suppress;   // Program Command to Suppress Low-Low Alarm
   PCmd_LoLoUnsuppress : ALIAS FOR LoLo.PCmd_Unsuppress;   // Program Command to Unsuppress Low-Low Alarm
   PCmd_LoLoUnshelve : ALIAS FOR LoLo.PCmd_Unshelve;   // Program Command to Unshelve Low-Low Alarm
   PCmd_FailAck : ALIAS FOR Fail.PCmd_Ack;   // Program Command to Acknowldege Analog Input Failure Alarm
   PCmd_FailSuppress : ALIAS FOR Fail.PCmd_Suppress;   // Program Command to Suppress Analog Input Failure Alarm
   PCmd_FailUnsuppress : ALIAS FOR Fail.PCmd_Unsuppress;   // Program Command to Unsuppress Analog Input Failure Alarm
   PCmd_FailUnshelve : ALIAS FOR Fail.PCmd_Unshelve;   // Program Command to Unshelve Analog Input Failure Alarm
END_VAR
VAR_OUTPUT
   Val : REAL; {access Read Only, visible}   // Analog Value (after Substitute PV, if used)
   Val_InpPV : REAL; {access Read Only, visible}   // Analog Input Value (actual, before Substitute PV selection)
   Val_PVMinCapt : REAL := 1.5e+38; {access Read Only}   // Captured PV Minimum (excursion) since last cleared
   Val_PVMaxCapt : REAL := -1.5e+38; {access Read Only}   // Captured PV Maximum (excursion) since last cleared
   Val_PVEUMin : REAL; {access Read Only}   // Minimum of scaled range = MIN (Cfg_PVEUMin, Cfg_PVEUMax)
   Val_PVEUMax : REAL := 100.0; {access Read Only}   // Maximum of scaled range = MAX (Cfg_PVEUMin, Cfg_PVEUMax)
   SrcQ_IO : DINT; {access Read Only}   // Source and Quality of primary I/O (enumeration)
   SrcQ : DINT; {access Read Only}   // Source and Quality of primary Val/Sts (enumeration)
   Val_Fault : DINT; {access Read Only}   // Device Fault Status 0=none, 20=Lo, 21=Hi, 24=LoLo, 25=HiHi, 32=Fail, 34=CfgErr
   Val_NotifyAll : DINT; {access Read Only}   // Highest Alarm prio and ack status this object + channel (enum)
   Val_UnackAlmC : DINT; {access Read Only}   // Count of Unacknowledged Alarms
   Sts_SubstPV : BOOL; {access Read Only}   // 1=Using Substitute PV (overrides input), 0=Using live Input PV from device
   Sts_PVBad : BOOL; {access Read Only}   // 1=PV Bad quality or Out of Range
   Sts_PVUncertain : BOOL; {access Read Only}   // 1=PV Value is Uncertain (quality)
   Sts_MaintByp : BOOL; {access Read Only}   // 1=A Maintenance Bypass is Active, display icon
   Sts_AlmInh : BOOL; {access Read Only}   // 1=An Alarm is Shelved, Disabled or Suppressed: display icon
   Sts_Err : BOOL; {access Read Only, visible}   // 1=Error in Config (see detail Err_ bits for reason), display icon
   Err_Raw : BOOL; {access Read Only}   // 1=Error in Config: Raw Input Scaling Min = Max
   Err_EU : BOOL; {access Read Only}   // 1=Error in Config: Scaled EU Min = Max
   Err_Timer : BOOL; {access Read Only}   // 1=Error in Config: On Delay, Off Delay, Gate Delay Time Invalid (use 0 to 2147483 s)
   Err_Filt : BOOL; {access Read Only}   // 1=Error in Config: PV filter params (RateTime, TC)
   Err_Alarm : BOOL; {access Read Only}   // 1=Error in Config: Alarm Min On Time, Shelf Time, Severity
   Sts_RdyReset : ALIAS FOR ORdy_Reset; {access Read Only}   // 1=A latched alarm or shed condition is ready to be reset
   Sts_RdyAck : BOOL; {access Read Only}   // 1=An alarm is ready to be acknowledged
   Sts_HiHiCmp : ALIAS FOR HiHiGate.Inp;   // PV High-High comparison result 1=High-High
   Sts_HiHiGate : ALIAS FOR HiHiGate.Sts_Gate; {access Read Only}   // PV High-High Gate Delay Status, 1=done
   Sts_HiHi : ALIAS FOR HiHi.Inp; {visible}   // 1=Analog Input is above High-High limit
   Alm_HiHi : ALIAS FOR HiHi.Alm;   // 1=Analog Input is in High-High Alarm
   Ack_HiHi : ALIAS FOR HiHi.Ack;   // 1=High-High Alarm has been acknowledged
   Sts_HiHiDisabled : ALIAS FOR HiHi.Disabled;   // 1=High-High Alarm has been Disabled by Maintenancy
   Sts_HiHiSuppressed : ALIAS FOR HiHi.Suppressed;   // 1=High-High Alarm has been Suppressed by Program
   Sts_HiHiShelved : ALIAS FOR HiHi.Shelved;   // 1=High-High Alarm has been Shelved by Operator
   Sts_HiCmp : ALIAS FOR HiGate.Inp;   // PV High comparison result 1=High
   Sts_HiGate : ALIAS FOR HiGate.Sts_Gate; {access Read Only}   // PV High Gate Delay Status, 1=done
   Sts_Hi : ALIAS FOR Hi.Inp; {visible}   // 1=Analog Input is above High limit
   Alm_Hi : ALIAS FOR Hi.Alm;   // 1=Analog Input is in High Alarm
   Ack_Hi : ALIAS FOR Hi.Ack;   // 1=High Alarm has been acknowledged
   Sts_HiDisabled : ALIAS FOR Hi.Disabled;   // 1=High Alarm has been Disabled by Maintenance
   Sts_HiSuppressed : ALIAS FOR Hi.Suppressed;   // 1=High Alarm has been Suppressed by Program
   Sts_HiShelved : ALIAS FOR Hi.Shelved;   // 1=High Alarm has been Shelved by Operator
   Sts_LoCmp : ALIAS FOR LoGate.Inp;   // PV Low comparison result 1=Low
   Sts_LoGate : ALIAS FOR LoGate.Sts_Gate; {access Read Only}   // PV Low Gate Delay Status, 1=done
   Sts_Lo : ALIAS FOR Lo.Inp; {visible}   // 1=Analog Input is below Low limit
   Alm_Lo : ALIAS FOR Lo.Alm;   // 1=Analog Input is in Low Alarm
   Ack_Lo : ALIAS FOR Lo.Ack;   // 1=Low Alarm has been acknowledged
   Sts_LoDisabled : ALIAS FOR Lo.Disabled;   // 1=Low Alarm has been Disabled by Maintenance
   Sts_LoSuppressed : ALIAS FOR Lo.Suppressed;   // 1=Low Alarm has been Suppressed by Program
   Sts_LoShelved : ALIAS FOR Lo.Shelved;   // 1=Low Alarm has been Shelved by Operator
   Sts_LoLoCmp : ALIAS FOR LoLoGate.Inp;   // PV Low-Low comparison result 1=Low-Low
   Sts_LoLoGate : ALIAS FOR LoLoGate.Sts_Gate; {access Read Only}   // PV Low-Low Gate Delay Status, 1=done
   Sts_LoLo : ALIAS FOR LoLo.Inp; {visible}   // 1=Analog Input is below Low-Low limit
   Alm_LoLo : ALIAS FOR LoLo.Alm;   // 1=Analog Input is in Low-Low Alarm
   Ack_LoLo : ALIAS FOR LoLo.Ack;   // 1=Low-Low Alarm has been acknowledged
   Sts_LoLoDisabled : ALIAS FOR LoLo.Disabled;   // 1=Low-Low Alarm has been Disabled by Maintenance
   Sts_LoLoSuppressed : ALIAS FOR LoLo.Suppressed;   // 1=Low-Low Alarm has been Suppressed by Program
   Sts_LoLoShelved : ALIAS FOR LoLo.Shelved;   // 1=Low-Low Alarm has been Shelved by Operator
   Sts_FailCmp : ALIAS FOR FailGate.Inp;   // PV Fail comparison result 1=Out of Range
   Sts_FailGate : ALIAS FOR FailGate.Sts_Gate; {access Read Only}   // PV Fail Gate Delay Status, 1=done
   Sts_Fail : ALIAS FOR Fail.Inp; {visible}   // 1=Analog Input is Out of Range or PV Bad
   Alm_Fail : ALIAS FOR Fail.Alm;   // 1=Analog Input Failure Alarm (PV Bad or Out of Range)
   Ack_Fail : ALIAS FOR Fail.Ack;   // 1=Analog Input Failure Alarm has been acknowledged
   Sts_FailDisabled : ALIAS FOR Fail.Disabled;   // 1=Analog input Failure Alarm has been Disabled by Maintenance
   Sts_FailSuppressed : ALIAS FOR Fail.Suppressed;   // 1=Analog Input Failure Alarm has been Suppressed by Program
   Sts_FailShelved : ALIAS FOR Fail.Shelved; {visible}   // 1=Analog Input Failure Alarm has been Shelved by Operator
   P_AIn : BOOL;   // Unique Parameter Name for auto - discovery
END_VAR
VAR
   LoLo : P_Alarm := (Cfg_AckReqd := 1, Cfg_AllowShelve := 1, Cfg_AllowDisable := 1, Cfg_Severity := 750, Cfg_AlmMinOnT := 5, PCfg_AllowExist := 1, Ack := 1);   // Low-Low Alarm
   Lo : P_Alarm := (Cfg_AckReqd := 1, Cfg_AllowShelve := 1, Cfg_AllowDisable := 1, Cfg_Severity := 500, Cfg_AlmMinOnT := 5, PCfg_AllowExist := 1, Ack := 1);   // Low Alarm
   Hi : P_Alarm := (Cfg_AckReqd := 1, Cfg_AllowShelve := 1, Cfg_AllowDisable := 1, Cfg_Severity := 500, Cfg_AlmMinOnT := 5, PCfg_AllowExist := 1, Ack := 1);   // High Alarm
   HiHi : P_Alarm := (Cfg_AckReqd := 1, Cfg_AllowShelve := 1, Cfg_AllowDisable := 1, Cfg_Severity := 750, Cfg_AlmMinOnT := 5, PCfg_AllowExist := 1, Ack := 1);   // High-High Alarm
   Cfg_EU : STRING_8 := '%';   // Engineering Units for display on HMI
   Cfg_Tag : STRING_20 := 'P_AIn';   // Tagname for display on HMI
   Cfg_Label : STRING_20 := 'Analog Input';   // Label for graphic symbol displayed on HMI
   Cfg_Desc : STRING_40 := 'Analog Input';   // Description for display on HMI
   Fail : P_Alarm := (Cfg_AckReqd := 1, Cfg_AllowShelve := 1, Cfg_AllowDisable := 1, Cfg_Severity := 1000, Cfg_AlmMinOnT := 5, PCfg_AllowExist := 1, Ack := 1);   // Analog Input Failure Alarm (bad quality or out of range)
   Wrk_Notify : DINT; {access None}   // Buffer for building Val_Notify
   HMI_Tab : SINT;   // Tab to display (FTView ME)
   Wrk_Fault : DINT; {access None}   // Buffer for building Val_Fault
   Wrk_SrcQ : DINT; {access None}   // Register for building Source / Quality enumeration
   Wrk_SubstPV : BOOL; {access None}   // Internal flag: Using Substitute PV
   Wrk_UnfiltPV : REAL; {access None}   // Unfiltered PV, input to 1st order filter
   Wrk_Alpha : REAL; {access None}   // Filter multiplier = (1 / (1+TC/dT) )
   Wrk_ScanT : TIMER := (PRE := 2147483647); {access None}   // Scan Timer (milliseconds, always runs)
   Wrk_ScanTime : REAL; {access None}   // Time since this instance was last scanned
   Wrk_FiltPV : REAL; {access None}   // Filtered PV
   Wrk_ValidONS : BOOL; {access None}   // Selected PV goes from Infinite or Not a Number to VALID
   Wrk_SelPVDINT : DINT; {access None}   // Selected PV check for Infinite or Non A Number
   Wrk_SelPVInfNaN : BOOL; {access None}   // Selected PV (Input or Substitute) is Infinite or NaN
   HMI_Type : STRING_16 := 'P_AIn'; {access Read Only}   // Must contain AOI name, used for HMI and Information S/W
   Wrk_Fail : BOOL; {access None}   // Internal flag: Fail Status
   Wrk_LoLo : BOOL; {access None}   // Internal flag: Low-Low Status
   Wrk_Lo : BOOL; {access None}   // Internal flag: Low Status
   Wrk_Hi : BOOL; {access None}   // Internal flag: High Status
   Wrk_HiHi : BOOL; {access None}   // Internal flag: High-High Status
   FailGate : P_Gate := (Inp_Gate := 1);   // Fail Alarm Gate / Delay Block
   LoLoGate : P_Gate := (Inp_Gate := 1);   // Low-Low Alarm Gate / Delay Block
   LoGate : P_Gate := (Inp_Gate := 1);   // Low Alarm Gate / Delay Block
   HiHiGate : P_Gate := (Inp_Gate := 1);   // High-High Alarm Gate / Delay Block
   HiGate : P_Gate := (Inp_Gate := 1);   // High Alarm Gate / Delay Block
   Wrk_InpInfNaN : BOOL; {access None}   // Input is Infinite or Not a Number
   Wrk_InpDINT : DINT; {access None}   // Input REAL bit pattern as a DINT (check for Inf/NaN)
   HMI_Lib : STRING_12 := 'RA-BAS'; {access Read Only}   // Display Library for Faceplate call-up
   Wrk_UnackAlmC : DINT; {access None}   // Buffer for building Val_UnackAlmC
   Val_Notify : DINT; {access Read Only}   // Highest Alarm prio and ack status this object only (enum)
   Cfg_Area : STRING_Area := 'area01';   // Process Area for security
   ORdy_ResetAckAll : BOOL; {access Read Only}   // 1=Ready for OCmd_ResetAckAll (enables HMI button)
   ORdy_Reset : BOOL; {access Read Only}   // 1=Ready for OCmd_Reset (enables HMI button)
   OCmd_ResetAckAll : BOOL;   // Operator Command to Reset and Acknowledge all Alarms
   OCmd_Reset : BOOL;   // Operator Command to Reset all Alarms requiring Reset
   OCmd_ClearCapt : BOOL;   // Operator Command to Clear the captured min / max PV excursion values
   MCmd_InpPV : BOOL;   // Maintenance Command to use Input PV (normal)
   MCmd_SubstPV : BOOL;   // Maintenance Command to use Substitute PV (override input)
   MRdy_InpPV : BOOL; {access Read Only}   // 1=Ready for MCmd_InpPV (enables HMI button)
   MRdy_SubstPV : BOOL; {access Read Only}   // 1=Ready for MCmd_SubstPV (enables HMI button)
   MSet_SubstPV : REAL;   // Maintenance-Entered Substitute PV (EU)
   Wrk_RawPV : REAL; {access None}   // Value of raw PV to be used for Out of Range checking
END_VAR

ROUTINE EnableInFalse   (* ladder *)
// Off-Scan: no Val update or alarm checking.  PV Bad Quality ("stale") is asserted.
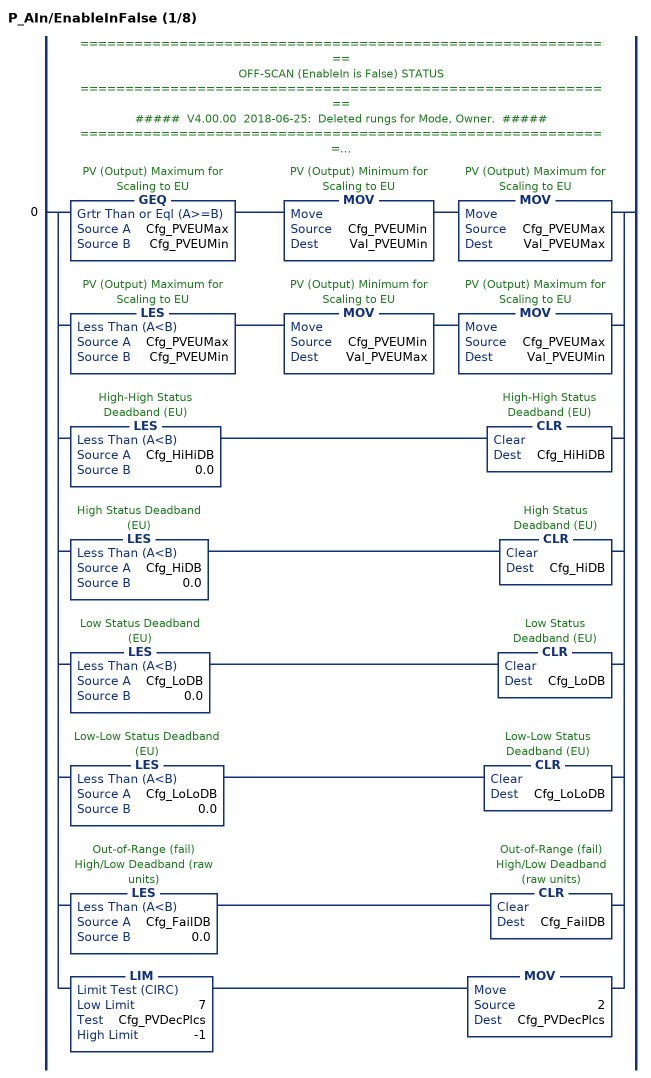
   // ============================================================
   // OFF-SCAN (EnableIn is False) STATUS
   // ============================================================
   // #####  V4.00.00  2018-06-25:  Deleted rungs for Mode, Owner.  #####
   // ============================================================
   // CONFIGURATION
   // ============================================================
   // This rung publishes the Values for the scaled range.
   // If this instruction is reverse scaled by reversing the scaled (EU) min and max configurations,
   // the values are swapped so the the EUMax Value is always greater than the EUMin Value.
   // This makes the HMI bargraph and trend coding easier, and provides values
   // that can be pinned to the configuration of a PID, so the AIn and PID ranges are in lockste
   // #####  V4.00.00  2018-06-25:  Added configurable decimal places for display on HMI.  #####
   // #####  Removed Err_DB, code ensures Status Deadband configs are always valid.  #####
   0: [GEQ(Cfg_PVEUMax,Cfg_PVEUMin) MOV(Cfg_PVEUMin,Val_PVEUMin) MOV(Cfg_PVEUMax,Val_PVEUMax) ,LES(Cfg_PVEUMax,Cfg_PVEUMin) MOV(Cfg_PVEUMin,Val_PVEUMax) MOV(Cfg_PVEUMax,Val_PVEUMin) ,LES(Cfg_HiHiDB,0.0) CLR(Cfg_HiHiDB) ,LES(Cfg_HiDB,0.0) CLR(Cfg_HiDB) ,LES(Cfg_LoDB,0.0) CLR(Cfg_LoDB) ,LES(Cfg_LoLoDB,0.0) CLR(Cfg_LoLoDB) ,LES(Cfg_FailDB,0.0) CLR(Cfg_FailDB) ,LIM(7,Cfg_PVDecPlcs,-1) MOV(2,Cfg_PVDecPlcs) ];
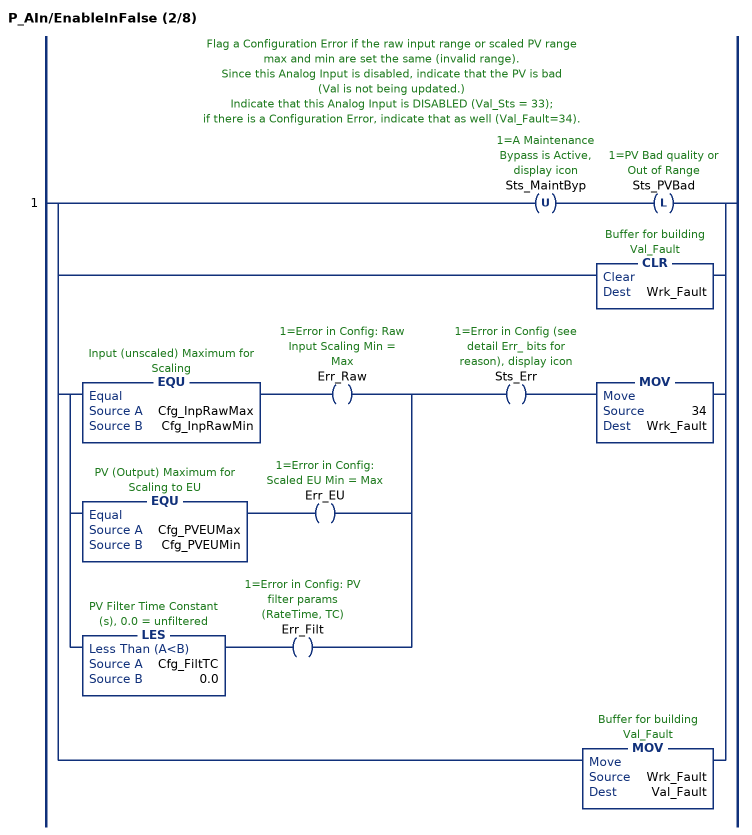
   // Flag a Configuration Error if the raw input range or scaled PV range
   // max and min are set the same (invalid range).
   // Since this Analog Input is disabled, indicate that the PV is bad
   // (Val is not being updated.)
   // Indicate that this Analog Input is DISABLED (Val_Sts = 33);
   // if there is a Configuration Error, indicate that as well (Val_Fault=34).
   1: [OTU(Sts_MaintByp) OTL(Sts_PVBad) ,CLR(Wrk_Fault) ,[EQU(Cfg_InpRawMax,Cfg_InpRawMin) OTE(Err_Raw) ,EQU(Cfg_PVEUMax,Cfg_PVEUMin) OTE(Err_EU) ,LES(Cfg_FiltTC,0.0) OTE(Err_Filt) ] OTE(Sts_Err) MOV(34,Wrk_Fault) ,MOV(Wrk_Fault,Val_Fault) ];
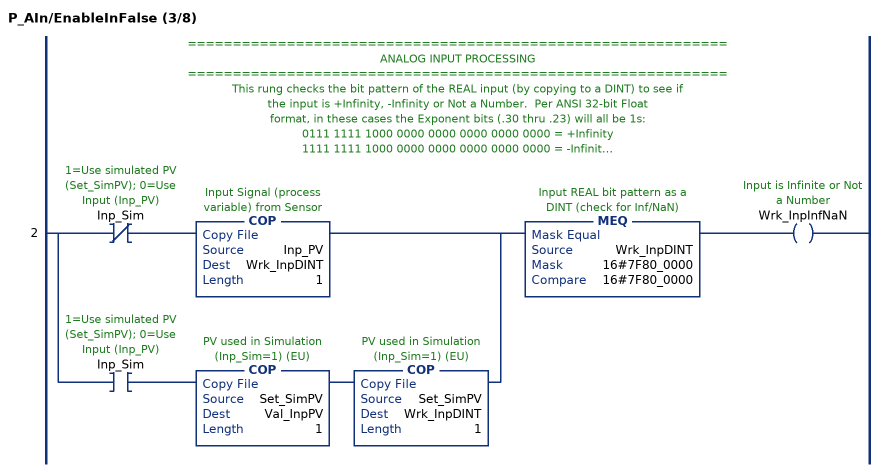
   // ============================================================
   // ANALOG INPUT PROCESSING
   // ============================================================
   // This rung checks the bit pattern of the REAL input (by copying to a DINT) to see if
   // the input is +Infinity, -Infinity or Not a Number.  Per ANSI 32-bit Float
   // format, in these cases the Exponent bits (.30 thru .23) will all be 1s:
   // 0111 1111 1000 0000 0000 0000 0000 0000 = +Infinity
   // 1111 1111 1000 0000 0000 0000 0000 0000 = -Infinity
   // x111 1111 1xxx xxxx xxxx xxxx xxxx xxxx = Not a Number
   2: [XIO(Inp_Sim) COP(Inp_PV,Wrk_InpDINT,1) ,XIC(Inp_Sim) COP(Set_SimPV,Val_InpPV,1) COP(Set_SimPV,Wrk_InpDINT,1) ]MEQ(Wrk_InpDINT,16#7F80_0000,16#7F80_0000)OTE(Wrk_InpInfNaN);
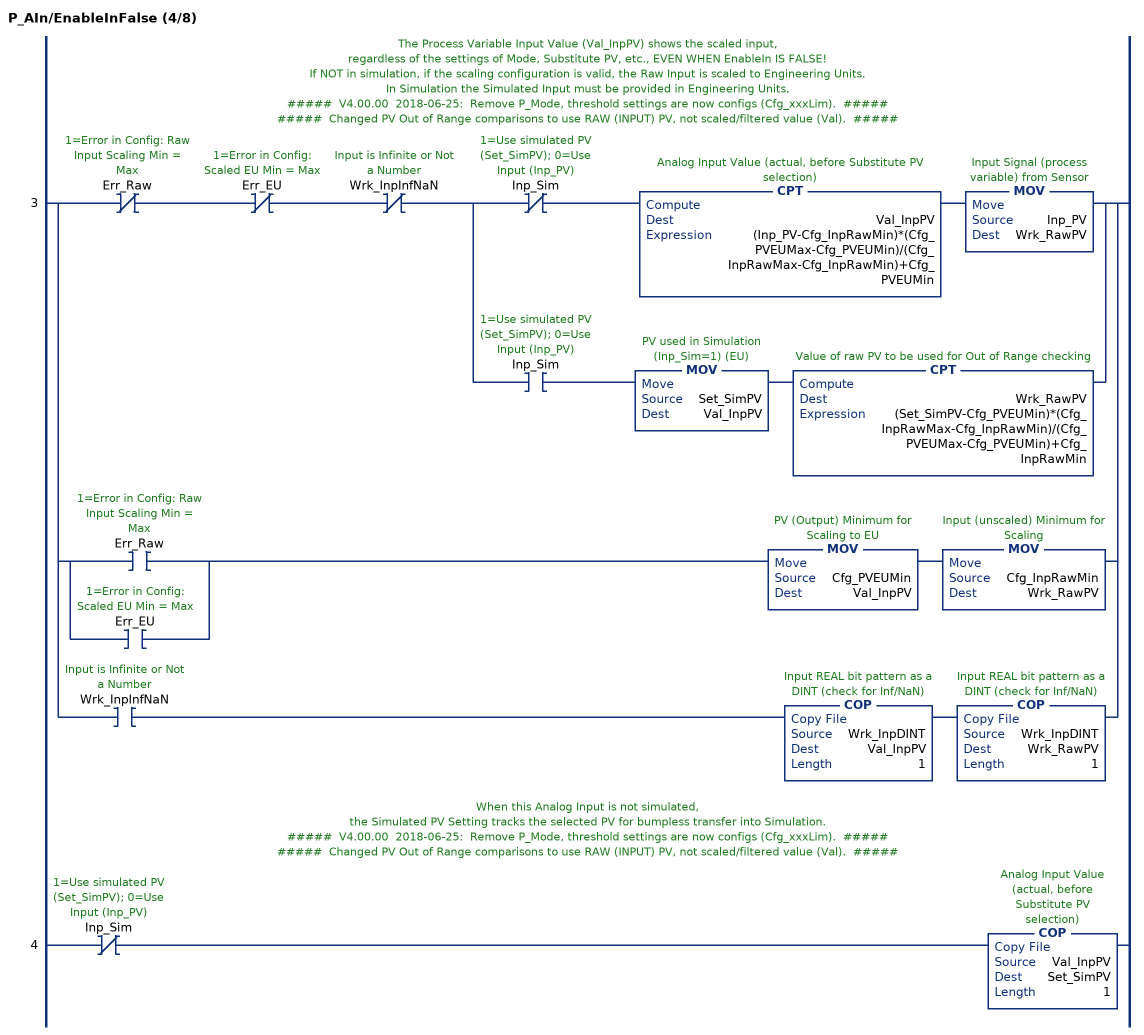
   // The Process Variable Input Value (Val_InpPV) shows the scaled input,
   // regardless of the settings of Mode, Substitute PV, etc., EVEN WHEN EnableIn IS FALSE!
   // If NOT in simulation, if the scaling configuration is valid, the Raw Input is scaled to Engineering Units.
   // In Simulation the Simulated Input must be provided in Engineering Units.
   // #####  V4.00.00  2018-06-25:  Remove P_Mode, threshold settings are now configs (Cfg_xxxLim).  #####
   // #####  Changed PV Out of Range comparisons to use RAW (INPUT) PV, not scaled/filtered value (Val).  #####
   3: [XIO(Err_Raw) XIO(Err_EU) XIO(Wrk_InpInfNaN) [XIO(Inp_Sim) CPT(Val_InpPV,(Inp_PV-Cfg_InpRawMin)*(Cfg_PVEUMax-Cfg_PVEUMin)/(Cfg_InpRawMax-Cfg_InpRawMin)+Cfg_PVEUMin) MOV(Inp_PV,Wrk_RawPV) ,XIC(Inp_Sim) MOV(Set_SimPV,Val_InpPV) CPT(Wrk_RawPV,(Set_SimPV-Cfg_PVEUMin)*(Cfg_InpRawMax-Cfg_InpRawMin)/(Cfg_PVEUMax-Cfg_PVEUMin)+Cfg_InpRawMin) ] ,[XIC(Err_Raw) ,XIC(Err_EU) ] MOV(Cfg_PVEUMin,Val_InpPV) MOV(Cfg_InpRawMin,Wrk_RawPV) ,XIC(Wrk_InpInfNaN) COP(Wrk_InpDINT,Val_InpPV,1) COP(Wrk_InpDINT,Wrk_RawPV,1) ];
   // When this Analog Input is not simulated,
   // the Simulated PV Setting tracks the selected PV for bumpless transfer into Simulation.
   // #####  V4.00.00  2018-06-25:  Remove P_Mode, threshold settings are now configs (Cfg_xxxLim).  #####
   // #####  Changed PV Out of Range comparisons to use RAW (INPUT) PV, not scaled/filtered value (Val).  #####
   4: XIO(Inp_Sim)COP(Val_InpPV,Set_SimPV,1);
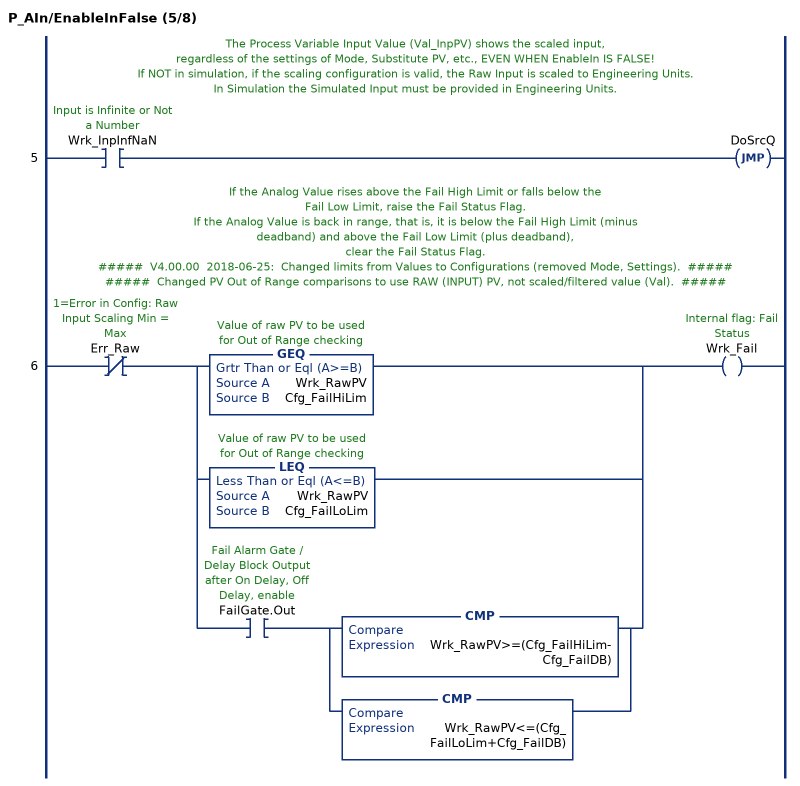
   // The Process Variable Input Value (Val_InpPV) shows the scaled input,
   // regardless of the settings of Mode, Substitute PV, etc., EVEN WHEN EnableIn IS FALSE!
   // If NOT in simulation, if the scaling configuration is valid, the Raw Input is scaled to Engineering Units.
   // In Simulation the Simulated Input must be provided in Engineering Units.
   5: XIC(Wrk_InpInfNaN)JMP(DoSrcQ);
   // If the Analog Value rises above the Fail High Limit or falls below the
   // Fail Low Limit, raise the Fail Status Flag.
   // If the Analog Value is back in range, that is, it is below the Fail High Limit (minus
   // deadband) and above the Fail Low Limit (plus deadband),
   // clear the Fail Status Flag.
   // #####  V4.00.00  2018-06-25:  Changed limits from Values to Configurations (removed Mode, Settings).  #####
   // #####  Changed PV Out of Range comparisons to use RAW (INPUT) PV, not scaled/filtered value (Val).  #####
   6: XIO(Err_Raw)[[GEQ(Wrk_RawPV,Cfg_FailHiLim) ,LEQ(Wrk_RawPV,Cfg_FailLoLim) ] ,XIC(FailGate.Out) [CMP(Wrk_RawPV>=(Cfg_FailHiLim-Cfg_FailDB)) ,CMP(Wrk_RawPV<=(Cfg_FailLoLim+Cfg_FailDB)) ] ]OTE(Wrk_Fail);
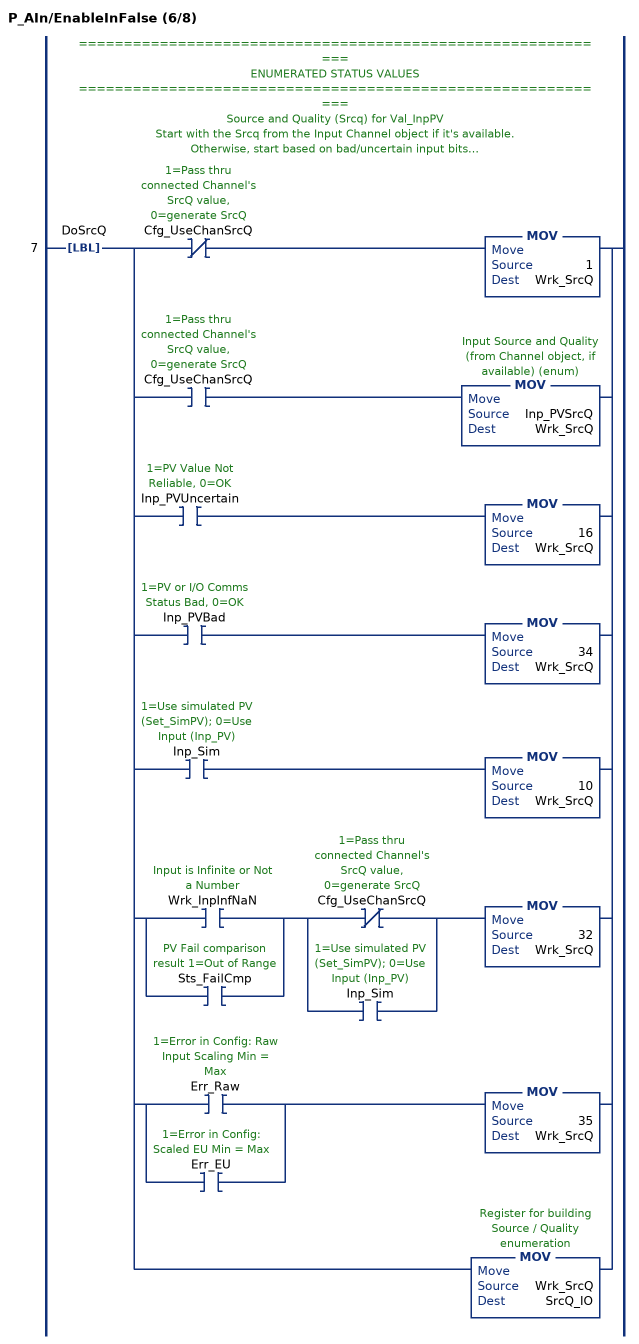
   // ============================================================
   // ENUMERATED STATUS VALUES
   // ============================================================
   // Source and Quality (Srcq) for Val_InpPV
   // Start with the Srcq from the Input Channel object if it's available.
   // Otherwise, start based on bad/uncertain input bits.
   // 0 = Good: live, confirmed good;   1 = Good: live, assumed good;
   // 2 = Good: no feedback, assumed good;   8 = Test: Simulated;   9 = Test: Loopback;
   // 10 = Test: Manually Entered;   16 = Uncertain: Live, off-spec;
   // 17 = Uncertain, Substituted at Device / Bus;   18 = Uncertain, Substituted at AOI;
   // 19 = Uncertain, using last known good;    20 = Uncertain, using replacement value;
   // 32 = Bad, Signal Failure;   33 = Bad, Channel Fault;
   // 34 = Bad, Module / Comms Fault;   35 = Bad, Invalid Configuration
   // #####  V4.00.00  2018-06-25:  Modified to correct precedence and value of Simulated PV.  #####
   // #####  V4.00.01  2018-08-29:  Modified handling of Simulated PV and scaling config errors.  #####
   7: LBL(DoSrcQ)[XIO(Cfg_UseChanSrcQ) MOV(1,Wrk_SrcQ) ,XIC(Cfg_UseChanSrcQ) MOV(Inp_PVSrcQ,Wrk_SrcQ) ,XIC(Inp_PVUncertain) MOV(16,Wrk_SrcQ) ,XIC(Inp_PVBad) MOV(34,Wrk_SrcQ) ,XIC(Inp_Sim) MOV(10,Wrk_SrcQ) ,[XIC(Wrk_InpInfNaN) ,XIC(Sts_FailCmp) ] [XIO(Cfg_UseChanSrcQ) ,XIC(Inp_Sim) ] MOV(32,Wrk_SrcQ) ,[XIC(Err_Raw) ,XIC(Err_EU) ] MOV(35,Wrk_SrcQ) ,MOV(Wrk_SrcQ,SrcQ_IO) ];
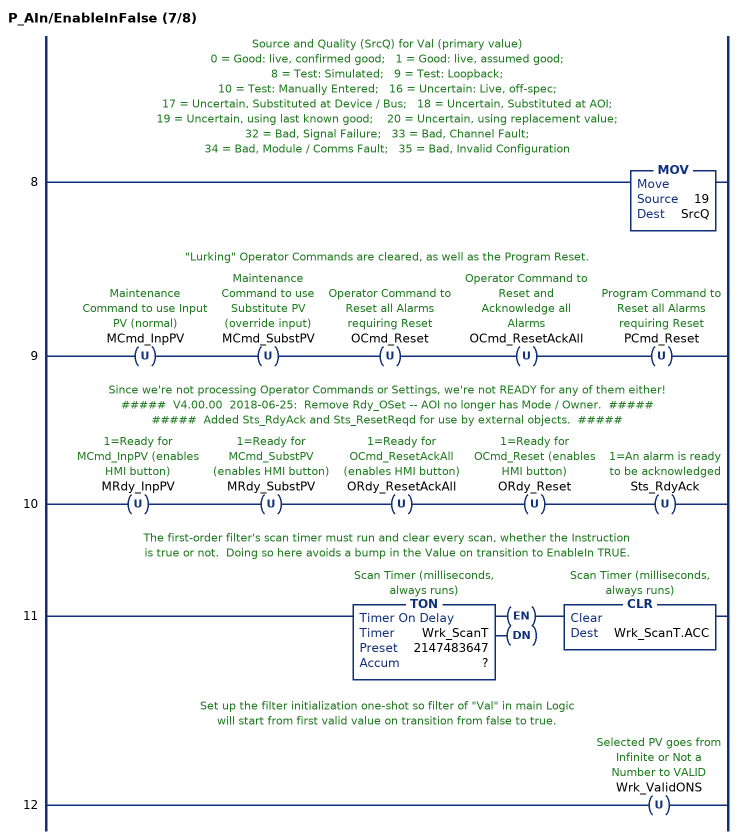
   // Source and Quality (SrcQ) for Val (primary value)
   // 0 = Good: live, confirmed good;   1 = Good: live, assumed good;
   // 8 = Test: Simulated;   9 = Test: Loopback;
   // 10 = Test: Manually Entered;   16 = Uncertain: Live, off-spec;
   // 17 = Uncertain, Substituted at Device / Bus;   18 = Uncertain, Substituted at AOI;
   // 19 = Uncertain, using last known good;    20 = Uncertain, using replacement value;
   // 32 = Bad, Signal Failure;   33 = Bad, Channel Fault;
   // 34 = Bad, Module / Comms Fault;   35 = Bad, Invalid Configuration
   8: MOV(19,SrcQ);
   // "Lurking" Operator Commands are cleared, as well as the Program Reset.
   9: OTU(MCmd_InpPV)OTU(MCmd_SubstPV)OTU(OCmd_Reset)OTU(OCmd_ResetAckAll)OTU(PCmd_Reset);
   // Since we're not processing Operator Commands or Settings, we're not READY for any of them either!
   // #####  V4.00.00  2018-06-25:  Remove Rdy_OSet -- AOI no longer has Mode / Owner.  #####
   // #####  Added Sts_RdyAck and Sts_ResetReqd for use by external objects.  #####
   10: OTU(MRdy_InpPV)OTU(MRdy_SubstPV)OTU(ORdy_ResetAckAll)OTU(ORdy_Reset)OTU(Sts_RdyAck);
   // The first-order filter's scan timer must run and clear every scan, whether the Instruction
   // is true or not.  Doing so here avoids a bump in the Value on transition to EnableIn TRUE.
   11: TON(Wrk_ScanT,?,?)CLR(Wrk_ScanT.ACC);
   // Set up the filter initialization one-shot so filter of "Val" in main Logic
   // will start from first valid value on transition from false to true.
   12: OTU(Wrk_ValidONS);
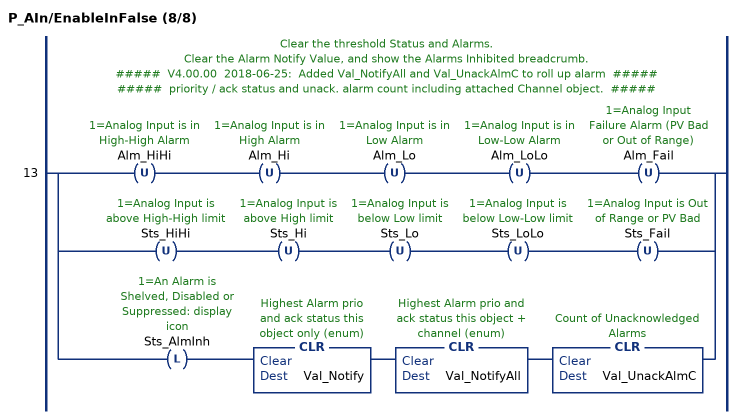
   // Clear the threshold Status and Alarms.
   // Clear the Alarm Notify Value, and show the Alarms Inhibited breadcrumb.
   // #####  V4.00.00  2018-06-25:  Added Val_NotifyAll and Val_UnackAlmC to roll up alarm  #####
   // #####  priority / ack status and unack. alarm count including attached Channel object.  #####
   13: [OTU(Alm_HiHi) OTU(Alm_Hi) OTU(Alm_Lo) OTU(Alm_LoLo) OTU(Alm_Fail) ,OTU(Sts_HiHi) OTU(Sts_Hi) OTU(Sts_Lo) OTU(Sts_LoLo) OTU(Sts_Fail) ,OTL(Sts_AlmInh) CLR(Val_Notify) CLR(Val_NotifyAll) CLR(Val_UnackAlmC) ];
END_ROUTINE

ROUTINE Logic   (* ladder *)
// Normal Scan - PV is scaled and alarms are generated
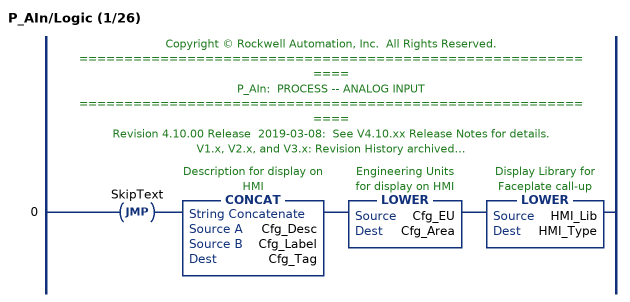
   // Copyright © Rockwell Automation, Inc.  All Rights Reserved.
   // ============================================================
   // P_AIn:  PROCESS -- ANALOG INPUT
   // ============================================================
   // Revision 4.10.00 Release  2019-03-08:  See V4.10.xx Release Notes for details.
   // V1.x, V2.x, and V3.x: Revision History archived.
   // V4.00.00  2018-06-25:  Removed P_Mode, PSet/Val_Owner and related OSets,
   //    PSets and Vals. Thresholds are now Cfgs. Changed Inf_ items to HMI_,
   // and added Cfg_Area for security. Added notify and unack count rollup for
   // Channel object. Changed Out-of-Range limit checks to use raw Input
   // (Inp_PV) instead of scaled PV (Val). (Changing EU scaling will not
   //    necessitate changing fail thresholds and deadband.)
   // Aligned ready bit naming with command bit names.
   // All OCmds/MCmds and ORdys/MRdys are now Local Tags.
   // Added Sts_RdyAck and Sts_ResetReqd for use by external objects.
   // Removed Err_DB, code ensures Status Deadband configs are always valid.
   // Added configurable decimal places for display on HMI.
   // V4.00.01  2018-08-29:  Modified handling of SrcQ_IO and SrcQ.
   // V4.10.00  2019-03-08:  Added Cfg_HasMoreObj.
   // ============================================================
   // This Instruction monitors an Analog Input from a flow, level, pressure,
   // temperature, or any other analog sensor, and provides:
   // *  Scaling, from Input (Raw) to PV (Engineering) Units
   // *  High-High, High, Low and Low-Low Status and Alarms, with Gate
   // inputs and configurable on-delay, off-delay and gate delay times
   // *  Monitoring of bad/uncertain PV status, floating point exceptions
   // and out-of-range conditions, with PV Fail alarm
   // *  Setting of a simulated input signal for process simulation
   // *  Capturing of the lowest and highest PV excursion values
   // *  Configurable status thresholds, threshold deadbands and out of range limits
   // *  Maintenance Commands to allow manual override of the input signal (Substitute PV)
   // Alarms are provided by P_Alarm AOI instances.
   // Status gating provided by P_Gate AOI instances.
   // ============================================================
   // SHOW LOCAL STRINGS
   // ============================================================
   // The STRINGs containing the text associated with each instance of this
   // instruction cannot be Input or Output Parameters, because STRINGs are not
   //  'atomic' types. (Inputs and Outputs must be SINT, INT, DINT, REAL, or BOOL.)
   // In order to make it easier to find and configure these STRINGs, this rung
   // was added.  THE JMP (and the LBL on the following rung)
   // MUST NOT BE REMOVED!!!
   // To view the STRINGs, go to the instruction instance (in LD or FBD), RIGHT-click
   // to bring up the context menu and select "Open Instruction Logic".
   // This rung will appear with the STRING values for the selected instance.
   // You may double-click the STRING values here to modify them as well.
   // #####  V4.00.00  2018-06-25:  Added string for Cfg_Area, renamed Inf_* to HMI_*.  #####
   // #####  Removed two rungs with Mode, Owner functions.  #####
   0: JMP(SkipText)CONCAT(Cfg_Desc,Cfg_Label,Cfg_Tag)LOWER(Cfg_EU,Cfg_Area)LOWER(HMI_Lib,HMI_Type);
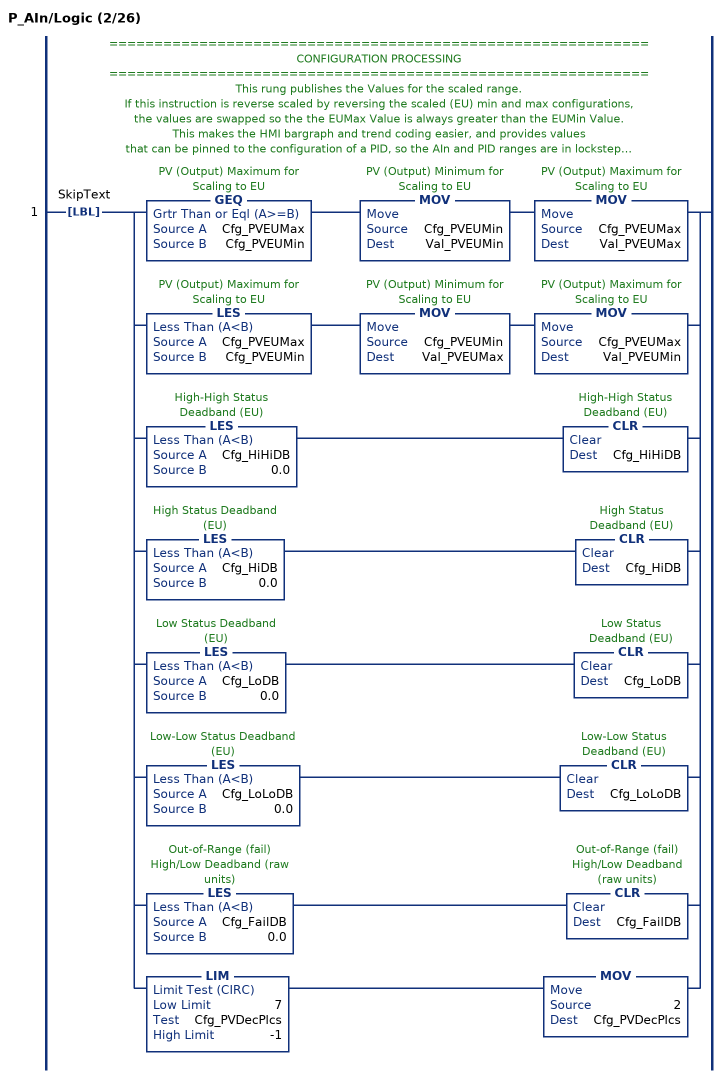
   // ============================================================
   // CONFIGURATION PROCESSING
   // ============================================================
   // This rung publishes the Values for the scaled range.
   // If this instruction is reverse scaled by reversing the scaled (EU) min and max configurations,
   // the values are swapped so the the EUMax Value is always greater than the EUMin Value.
   // This makes the HMI bargraph and trend coding easier, and provides values
   // that can be pinned to the configuration of a PID, so the AIn and PID ranges are in lockstep.
   // This rung also ensures valid entries for Status Threshold Deadband configs
   // and the number of decimal places for display of the PV.
   // #####  V4.00.00  2018-06-25:  Added configurable decimal places for display on HMI.  #####
   // #####  Removed Err_DB, code ensures Status Deadband configs are always valid.  #####
   1: LBL(SkipText)[GEQ(Cfg_PVEUMax,Cfg_PVEUMin) MOV(Cfg_PVEUMin,Val_PVEUMin) MOV(Cfg_PVEUMax,Val_PVEUMax) ,LES(Cfg_PVEUMax,Cfg_PVEUMin) MOV(Cfg_PVEUMin,Val_PVEUMax) MOV(Cfg_PVEUMax,Val_PVEUMin) ,LES(Cfg_HiHiDB,0.0) CLR(Cfg_HiHiDB) ,LES(Cfg_HiDB,0.0) CLR(Cfg_HiDB) ,LES(Cfg_LoDB,0.0) CLR(Cfg_LoDB) ,LES(Cfg_LoLoDB,0.0) CLR(Cfg_LoLoDB) ,LES(Cfg_FailDB,0.0) CLR(Cfg_FailDB) ,LIM(7,Cfg_PVDecPlcs,-1) MOV(2,Cfg_PVDecPlcs) ];
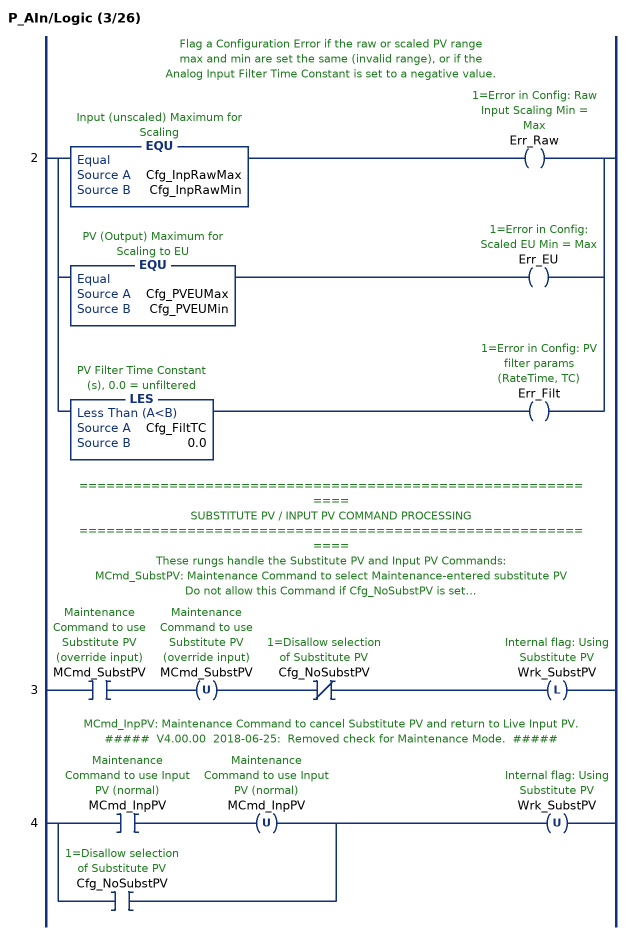
   // Flag a Configuration Error if the raw or scaled PV range
   // max and min are set the same (invalid range), or if the
   // Analog Input Filter Time Constant is set to a negative value.
   2: [EQU(Cfg_InpRawMax,Cfg_InpRawMin) OTE(Err_Raw) ,EQU(Cfg_PVEUMax,Cfg_PVEUMin) OTE(Err_EU) ,LES(Cfg_FiltTC,0.0) OTE(Err_Filt) ];
   // ============================================================
   // SUBSTITUTE PV / INPUT PV COMMAND PROCESSING
   // ============================================================
   // These rungs handle the Substitute PV and Input PV Commands:
   // MCmd_SubstPV: Maintenance Command to select Maintenance-entered substitute PV
   // Do not allow this Command if Cfg_NoSubstPV is set.
   // #####  V4.00.00  2018-06-25:  Removed check for Maintenance Mode.  #####
   3: XIC(MCmd_SubstPV)OTU(MCmd_SubstPV)XIO(Cfg_NoSubstPV)OTL(Wrk_SubstPV);
   // MCmd_InpPV: Maintenance Command to cancel Substitute PV and return to Live Input PV.
   // #####  V4.00.00  2018-06-25:  Removed check for Maintenance Mode.  #####
   4: [XIC(MCmd_InpPV) OTU(MCmd_InpPV) ,XIC(Cfg_NoSubstPV) ]OTU(Wrk_SubstPV);
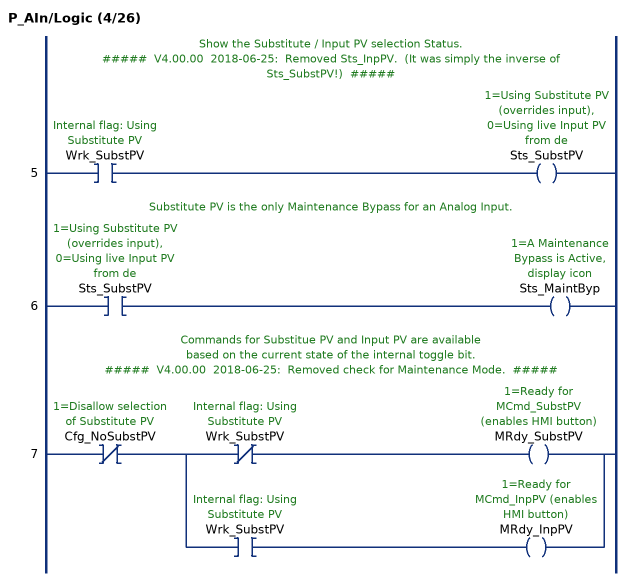
   // Show the Substitute / Input PV selection Status.
   // #####  V4.00.00  2018-06-25:  Removed Sts_InpPV.  (It was simply the inverse of Sts_SubstPV!)  #####
   5: XIC(Wrk_SubstPV)OTE(Sts_SubstPV);
   // Substitute PV is the only Maintenance Bypass for an Analog Input.
   6: XIC(Sts_SubstPV)OTE(Sts_MaintByp);
   // Commands for Substitue PV and Input PV are available
   // based on the current state of the internal toggle bit.
   // #####  V4.00.00  2018-06-25:  Removed check for Maintenance Mode.  #####
   7: XIO(Cfg_NoSubstPV)[XIO(Wrk_SubstPV) OTE(MRdy_SubstPV) ,XIC(Wrk_SubstPV) OTE(MRdy_InpPV) ];
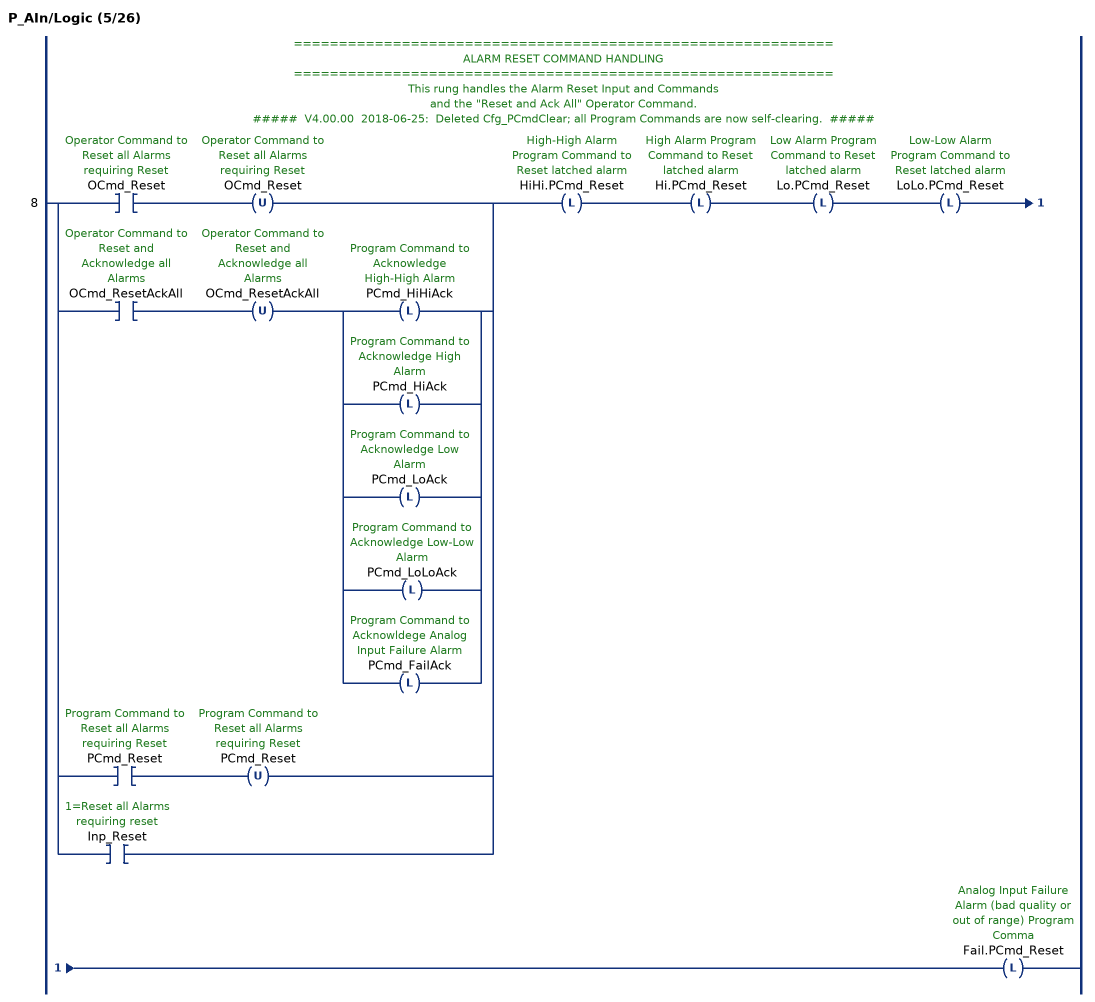
   // ============================================================
   // ALARM RESET COMMAND HANDLING
   // ============================================================
   // This rung handles the Alarm Reset Input and Commands
   // and the "Reset and Ack All" Operator Command.
   // #####  V4.00.00  2018-06-25:  Deleted Cfg_PCmdClear; all Program Commands are now self-clearing.  #####
   8: [XIC(OCmd_Reset) OTU(OCmd_Reset) ,XIC(OCmd_ResetAckAll) OTU(OCmd_ResetAckAll) [OTL(PCmd_HiHiAck) ,OTL(PCmd_HiAck) ,OTL(PCmd_LoAck) ,OTL(PCmd_LoLoAck) ,OTL(PCmd_FailAck) ] ,XIC(PCmd_Reset) OTU(PCmd_Reset) ,XIC(Inp_Reset) ]OTL(HiHi.PCmd_Reset)OTL(Hi.PCmd_Reset)OTL(Lo.PCmd_Reset)OTL(LoLo.PCmd_Reset)OTL(Fail.PCmd_Reset);
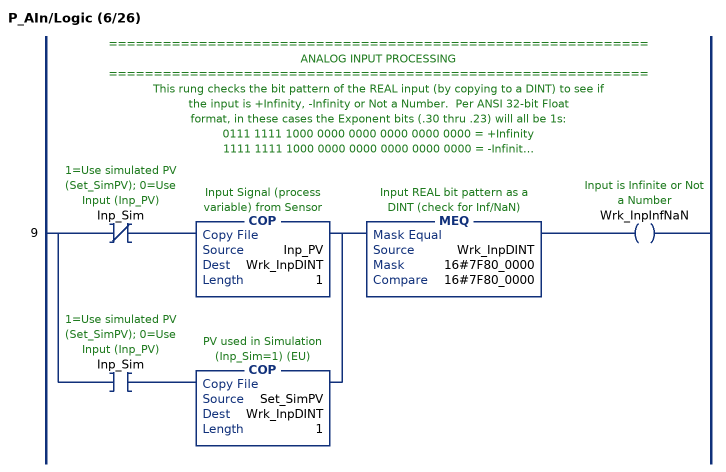
   // ============================================================
   // ANALOG INPUT PROCESSING
   // ============================================================
   // This rung checks the bit pattern of the REAL input (by copying to a DINT) to see if
   // the input is +Infinity, -Infinity or Not a Number.  Per ANSI 32-bit Float
   // format, in these cases the Exponent bits (.30 thru .23) will all be 1s:
   // 0111 1111 1000 0000 0000 0000 0000 0000 = +Infinity
   // 1111 1111 1000 0000 0000 0000 0000 0000 = -Infinity
   // x111 1111 1xxx xxxx xxxx xxxx xxxx xxxx = Not a Number
   9: [XIO(Inp_Sim) COP(Inp_PV,Wrk_InpDINT,1) ,XIC(Inp_Sim) COP(Set_SimPV,Wrk_InpDINT,1) ]MEQ(Wrk_InpDINT,16#7F80_0000,16#7F80_0000)OTE(Wrk_InpInfNaN);
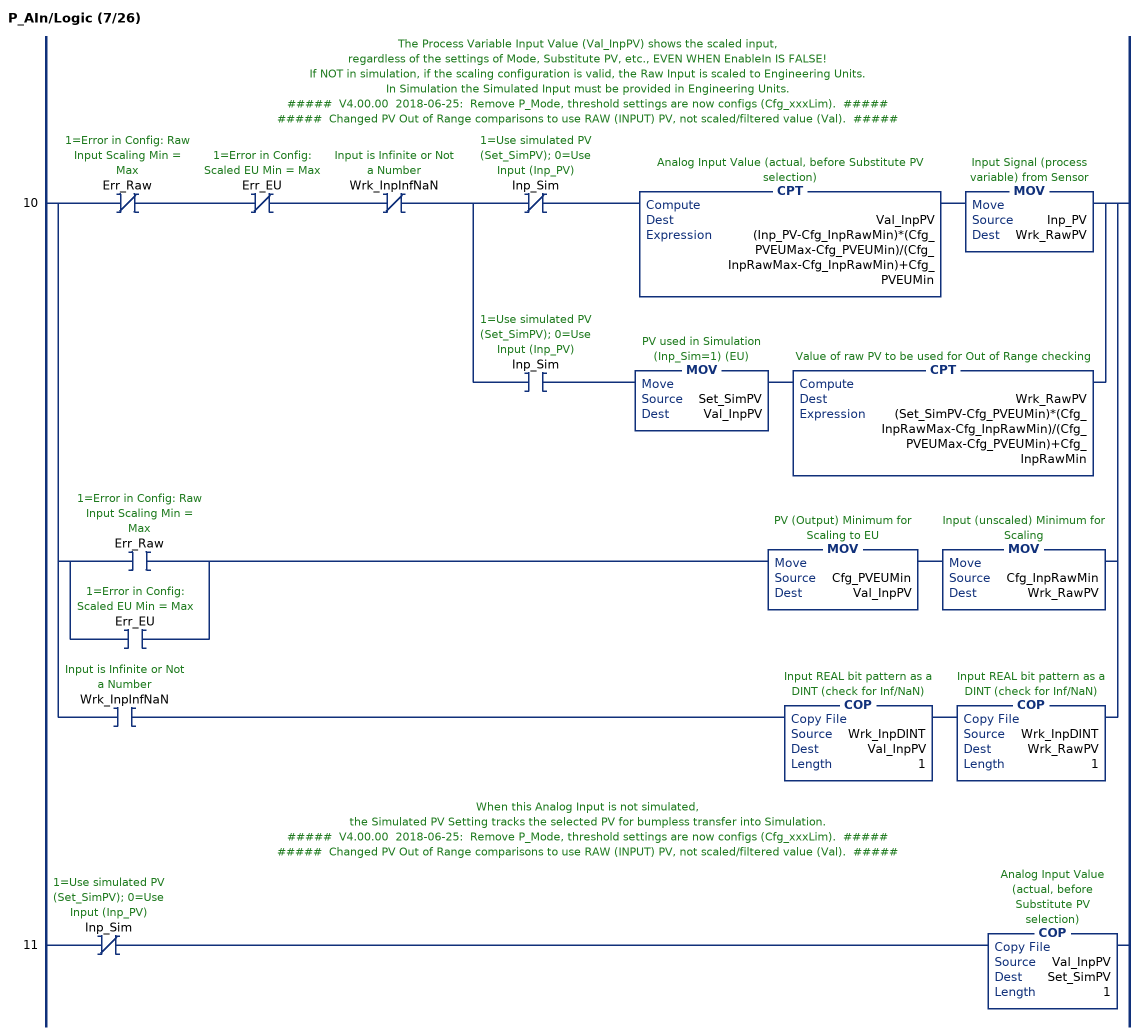
   // The Process Variable Input Value (Val_InpPV) shows the scaled input,
   // regardless of the settings of Mode, Substitute PV, etc., EVEN WHEN EnableIn IS FALSE!
   // If NOT in simulation, if the scaling configuration is valid, the Raw Input is scaled to Engineering Units.
   // In Simulation the Simulated Input must be provided in Engineering Units.
   // #####  V4.00.00  2018-06-25:  Remove P_Mode, threshold settings are now configs (Cfg_xxxLim).  #####
   // #####  Changed PV Out of Range comparisons to use RAW (INPUT) PV, not scaled/filtered value (Val).  #####
   10: [XIO(Err_Raw) XIO(Err_EU) XIO(Wrk_InpInfNaN) [XIO(Inp_Sim) CPT(Val_InpPV,(Inp_PV-Cfg_InpRawMin)*(Cfg_PVEUMax-Cfg_PVEUMin)/(Cfg_InpRawMax-Cfg_InpRawMin)+Cfg_PVEUMin) MOV(Inp_PV,Wrk_RawPV) ,XIC(Inp_Sim) MOV(Set_SimPV,Val_InpPV) CPT(Wrk_RawPV,(Set_SimPV-Cfg_PVEUMin)*(Cfg_InpRawMax-Cfg_InpRawMin)/(Cfg_PVEUMax-Cfg_PVEUMin)+Cfg_InpRawMin) ] ,[XIC(Err_Raw) ,XIC(Err_EU) ] MOV(Cfg_PVEUMin,Val_InpPV) MOV(Cfg_InpRawMin,Wrk_RawPV) ,XIC(Wrk_InpInfNaN) COP(Wrk_InpDINT,Val_InpPV,1) COP(Wrk_InpDINT,Wrk_RawPV,1) ];
   // When this Analog Input is not simulated,
   // the Simulated PV Setting tracks the selected PV for bumpless transfer into Simulation.
   // #####  V4.00.00  2018-06-25:  Remove P_Mode, threshold settings are now configs (Cfg_xxxLim).  #####
   // #####  Changed PV Out of Range comparisons to use RAW (INPUT) PV, not scaled/filtered value (Val).  #####
   11: XIO(Inp_Sim)COP(Val_InpPV,Set_SimPV,1);
